LIN {X 0,Y 368.879,Z 269.346,A -85,B 0,C 180,E1 -12556.695,E2 -12556.695} C_VEL
LIN {X 0,Y 368.88,Z 269.35,A -85,B 0,C 180,E1 -12559.648,E2 -12559.648} C_VEL
LIN {X 0,Y 368.892,Z 269.345,A -85,B 0,C 180,E1 -12563.145,E2 -12563.145} C_VEL
LIN {X 0,Y 368.891,Z 269.344,A -85,B 0,C 180,E1 -12566.461,E2 -12566.461} C_VEL
LIN {X 0,Y 368.891,Z 269.346,A -85,B 0,C 180,E1 -12569.043,E2 -12569.043} C_VEL
LIN {X 0,Y 368.902,Z 269.348,A -85,B 0,C 180,E1 -12571.557,E2 -12571.557} C_VEL
LIN {X 0,Y 368.909,Z 269.347,A -85,B 0,C 180,E1 -12575.221,E2 -12575.221} C_VEL
LIN {X 0,Y 368.904,Z 269.344,A -85,B 0,C 180,E1 -12578.779,E2 -12578.779} C_VEL
LIN {X 0,Y 368.948,Z 269.337,A -85,B 0,C 180,E1 -12582.255,E2 -12582.255} C_VEL
LIN {X 0,Y 369.032,Z 269.327,A -85,B 0,C 180,E1 -12586.228,E2 -12586.228} C_VEL
LIN {X 0,Y 369.052,Z 269.324,A -85,B 0,C 180,E1 -12590.131,E2 -12590.131} C_VEL
LIN {X 0,Y 369.15,Z 269.313,A -85,B 0,C 180,E1 -12593.441,E2 -12593.441} C_VEL
LIN {X 0,Y 369.295,Z 269.294,A -85,B 0,C 180,E1 -12597.819,E2 -12597.819} C_VEL
LIN {X 0,Y 369.295,Z 269.297,A -85,B 0,C 180,E1 -12602.181,E2 -12602.181} C_VEL
LIN {X 0,Y 369.148,Z 269.316,A -85,B 0,C 180,E1 -12606.559,E2 -12606.559} C_VEL
LIN {X 0,Y 369.052,Z 269.326,A -85,B 0,C 180,E1 -12609.869,E2 -12609.869} C_VEL
LIN {X 0,Y 369.032,Z 269.329,A -85,B 0,C 180,E1 -12613.772,E2 -12613.772} C_VEL
LIN {X 0,Y 368.948,Z 269.34,A -85,B 0,C 180,E1 -12617.745,E2 -12617.745} C_VEL
LIN {X 0,Y 368.903,Z 269.343,A -85,B 0,C 180,E1 -12621.221,E2 -12621.221} C_VEL
LIN {X 0,Y 368.902,Z 269.348,A -85,B 0,C 180,E1 -12623.874,E2 -12623.874} C_VEL
LIN {X 0,Y 368.851,Z 269.35,A -85,B 0,C 180,E1 -12627.212,E2 -12627.212} C_VEL
LIN {X 0,Y 368.886,Z 269.35,A -85,B 0,C 180,E1 -12629.693,E2 -12629.693} C_VEL
LIN {X 0,Y 368.89,Z 269.345,A -85,B 0,C 180,E1 -12633.043,E2 -12633.043} C_VEL
LIN {X 0,Y 368.91,Z 269.342,A -85,B 0,C 180,E1 -12636.198,E2 -12636.198} C_VEL
LIN {X 0,Y 368.868,Z 269.349,A -85,B 0,C 180,E1 -12638.957,E2 -12638.957} C_VEL
LIN {X 0,Y 368.853,Z 269.349,A -85,B 0,C 180,E1 -12642.006,E2 -12642.006} C_VEL
LIN {X 0,Y 368.869,Z 269.353,A -85,B 0,C 180,E1 -12645.175,E2 -12645.175} C_VEL
LIN {X 0,Y 368.856,Z 269.348,A -85,B 0,C 180,E1 -12648.175,E2 -12648.175} C_VEL
LIN {X 0,Y 368.871,Z 269.349,A -85,B 0,C 180,E1 -12651.367,E2 -12651.367} C_VEL
LIN {X 0,Y 368.926,Z 269.343,A -85,B 0,C 180,E1 -12655.146,E2 -12655.146} C_VEL
LIN {X 0,Y 368.892,Z 269.347,A -85,B 0,C 180,E1 -12659.044,E2 -12659.044} C_VEL
LIN {X 0,Y 368.932,Z 269.441,A -85,B 0,C 180,E1 -12662.564,E2 -12662.564} C_VEL
LIN {X 0,Y 371.142,Z 280.964,A -85,B 0,C 180,E1 -12665.558,E2 -12665.558} C_VEL
LIN {X 0,Y 370.932,Z 287.523,A -85,B 0,C 180,E1 -12667.145,E2 -12667.145} C_VEL
LIN {X 0,Y 369.772,Z 303.185,A -85,B 0,C 180,E1 -12670.862,E2 -12670.862} C_VEL
LIN {X 0,Y 369.194,Z 312.035,A -85,B 0,C 180,E1 -12672.947,E2 -12672.947} C_VEL
LIN {X 0,Y 372.572,Z 338.491,A -85,B 0,C 180,E1 -12673.629,E2 -12673.629} C_VEL
LIN {X 0,Y 373.125,Z 345.859,A -85,B 0,C 180,E1 -12673.798,E2 -12673.798} C_VEL
LIN {X 0,Y 372.569,Z 389.778,A -85,B 0,C 180,E1 -12674.664,E2 -12674.664} C_VEL
LIN {X 0,Y 372.153,Z 399.376,A -85,B 0,C 180,E1 -12674.986,E2 -12674.986} C_VEL
LIN {X 0,Y 371.63,Z 409.413,A -85,B 0,C 180,E1 -12675.489,E2 -12675.489} C_VEL
LIN {X 0,Y 370.884,Z 420.823,A -85,B 0,C 180,E1 -12676.299,E2 -12676.299} C_VEL
LIN {X 0,Y 370.198,Z 429.423,A -85,B 0,C 180,E1 -12677.111,E2 -12677.111} C_VEL
LIN {X 0,Y 369.516,Z 437.52,A -85,B 0,C 180,E1 -12678.064,E2 -12678.064} C_VEL
LIN {X 0,Y 368.999,Z 444.218,A -85,B 0,C 180,E1 -12679.021,E2 -12679.021} C_VEL
LIN {X 0,Y 368.476,Z 450.579,A -85,B 0,C 180,E1 -12680.116,E2 -12680.116} C_VEL
LIN {X 0,Y 368.086,Z 455.87,A -85,B 0,C 180,E1 -12681.214,E2 -12681.214} C_VEL
LIN {X 0,Y 367.863,Z 460.289,A -85,B 0,C 180,E1 -12682.315,E2 -12682.315} C_VEL
LIN {X 0,Y 367.557,Z 465.239,A -85,B 0,C 180,E1 -12683.87,E2 -12683.87} C_VEL
LIN {X 0,Y 367.535,Z 468.17,A -85,B 0,C 180,E1 -12685.064,E2 -12685.064} C_VEL
LIN {X 0,Y 367.462,Z 471.098,A -85,B 0,C 180,E1 -12686.711,E2 -12686.711} C_VEL
LIN {X 0,Y 367.541,Z 472.367,A -85,B 0,C 180,E1 -12687.809,E2 -12687.809} C_VEL
LIN {X 0,Y 367.585,Z 473.154,A -85,B 0,C 180,E1 -12688.905,E2 -12688.905} C_VEL
LIN {X 0,Y 367.581,Z 473.451,A -85,B 0,C 180,E1 -12690.001,E2 -12690.001} C_VEL
LIN {X 0,Y 367.585,Z 473.151,A -85,B 0,C 180,E1 -12691.096,E2 -12691.096} C_VEL
LIN {X 0,Y 367.542,Z 472.355,A -85,B 0,C 180,E1 -12692.192,E2 -12692.192} C_VEL
LIN {X 0,Y 367.462,Z 471.079,A -85,B 0,C 180,E1 -12693.29,E2 -12693.29} C_VEL
LIN {X 0,Y 367.535,Z 468.144,A -85,B 0,C 180,E1 -12694.937,E2 -12694.937} C_VEL
LIN {X 0,Y 367.557,Z 465.207,A -85,B 0,C 180,E1 -12696.13,E2 -12696.13} C_VEL
LIN {X 0,Y 367.832,Z 460.241,A -85,B 0,C 180,E1 -12697.687,E2 -12697.687} C_VEL
LIN {X 0,Y 368.27,Z 453.362,A -85,B 0,C 180,E1 -12699.336,E2 -12699.336} C_VEL
LIN {X 0,Y 368.87,Z 445.856,A -85,B 0,C 180,E1 -12700.706,E2 -12700.706} C_VEL
LIN {X 0,Y 369.431,Z 438.457,A -85,B 0,C 180,E1 -12701.801,E2 -12701.801} C_VEL
LIN {X 0,Y 370.069,Z 430.542,A -85,B 0,C 180,E1 -12702.755,E2 -12702.755} C_VEL
LIN {X 0,Y 370.79,Z 422.188,A -85,B 0,C 180,E1 -12703.566,E2 -12703.566} C_VEL
LIN {X 0,Y 371.428,Z 411.508,A -85,B 0,C 180,E1 -12704.38,E2 -12704.38} C_VEL
LIN {X 0,Y 372.091,Z 399.889,A -85,B 0,C 180,E1 -12704.983,E2 -12704.983} C_VEL
LIN {X 0,Y 372.515,Z 390.149,A -85,B 0,C 180,E1 -12705.316,E2 -12705.316} C_VEL
LIN {X 0,Y 373.127,Z 345.225,A -85,B 0,C 180,E1 -12706.202,E2 -12706.202} C_VEL
LIN {X 0,Y 371.249,Z 327.242,A -85,B 0,C 180,E1 -12706.638,E2 -12706.638} C_VEL
LIN {X 0,Y 369.171,Z 312.021,A -85,B 0,C 180,E1 -12707.045,E2 -12707.045} C_VEL
LIN {X 0,Y 370.215,Z 297.109,A -85,B 0,C 180,E1 -12710.561,E2 -12710.561} C_VEL
LIN {X 0,Y 371.25,Z 282.618,A -85,B 0,C 180,E1 -12714.018,E2 -12714.018} C_VEL
LIN {X 0,Y 369.812,Z 273.814,A -85,B 0,C 180,E1 -12716.27,E2 -12716.27} C_VEL
LIN {X 0,Y 368.889,Z 269.349,A -85,B 0,C 180,E1 -12717.479,E2 -12717.479} C_VEL
LIN {X 0,Y 368.886,Z 269.348,A -85,B 0,C 180,E1 -12720.981,E2 -12720.981} C_VEL
LIN {X 0,Y 368.93,Z 269.342,A -85,B 0,C 180,E1 -12724.855,E2 -12724.855} C_VEL
LIN {X 0,Y 368.874,Z 269.348,A -85,B 0,C 180,E1 -12728.634,E2 -12728.634} C_VEL
LIN {X 0,Y 368.858,Z 269.348,A -85,B 0,C 180,E1 -12732.005,E2 -12732.005} C_VEL
LIN {X 0,Y 368.874,Z 269.348,A -85,B 0,C 180,E1 -12735.175,E2 -12735.175} C_VEL
LIN {X 0,Y 368.86,Z 269.349,A -85,B 0,C 180,E1 -12738.175,E2 -12738.175} C_VEL
LIN {X 0,Y 368.876,Z 269.346,A -85,B 0,C 180,E1 -12741.367,E2 -12741.367} C_VEL
LIN {X 0,Y 368.931,Z 269.34,A -85,B 0,C 180,E1 -12745.146,E2 -12745.146} C_VEL
LIN {X 0,Y 368.897,Z 269.344,A -85,B 0,C 180,E1 -12749.044,E2 -12749.044} C_VEL
LIN {X 0,Y 368.907,Z 269.342,A -85,B 0,C 180,E1 -12751.558,E2 -12751.558} C_VEL
LIN {X 0,Y 368.919,Z 269.344,A -85,B 0,C 180,E1 -12754.014,E2 -12754.014} C_VEL
LIN {X 0,Y 368.895,Z 269.345,A -85,B 0,C 180,E1 -12757.603,E2 -12757.603} C_VEL
LIN {X 0,Y 368.898,Z 269.343,A -85,B 0,C 180,E1 -12761.103,E2 -12761.103} C_VEL
LIN {X 0,Y 368.921,Z 269.341,A -85,B 0,C 180,E1 -12764.532,E2 -12764.532} C_VEL
LIN {X 0,Y 369.024,Z 269.327,A -85,B 0,C 180,E1 -12766.789,E2 -12766.789} C_VEL
LIN {X 0,Y 369.058,Z 269.326,A -85,B 0,C 180,E1 -12770.132,E2 -12770.132} C_VEL
LIN {X 0,Y 369.156,Z 269.315,A -85,B 0,C 180,E1 -12773.441,E2 -12773.441} C_VEL
LIN {X 0,Y 369.297,Z 269.297,A -85,B 0,C 180,E1 -12777.819,E2 -12777.819} C_VEL
LIN {X 0,Y 369.302,Z 269.293,A -85,B 0,C 180,E1 -12782.181,E2 -12782.181} C_VEL
LIN {X 0,Y 369.156,Z 269.312,A -85,B 0,C 180,E1 -12786.559,E2 -12786.559} C_VEL
LIN {X 0,Y 369.059,Z 269.324,A -85,B 0,C 180,E1 -12789.869,E2 -12789.869} C_VEL
LIN {X 0,Y 369.039,Z 269.326,A -85,B 0,C 180,E1 -12793.772,E2 -12793.772} C_VEL
LIN {X 0,Y 368.955,Z 269.336,A -85,B 0,C 180,E1 -12797.745,E2 -12797.745} C_VEL
LIN {X 0,Y 368.91,Z 269.344,A -85,B 0,C 180,E1 -12801.221,E2 -12801.221} C_VEL
LIN {X 0,Y 368.91,Z 269.342,A -85,B 0,C 180,E1 -12803.874,E2 -12803.874} C_VEL
LIN {X 0,Y 368.86,Z 269.349,A -85,B 0,C 180,E1 -12807.212,E2 -12807.212} C_VEL
LIN {X 0,Y 368.894,Z 269.344,A -85,B 0,C 180,E1 -12809.692,E2 -12809.692} C_VEL
LIN {X 0,Y 368.898,Z 269.344,A -85,B 0,C 180,E1 -12813.043,E2 -12813.043} C_VEL
LIN {X 0,Y 368.913,Z 269.346,A -85,B 0,C 180,E1 -12816.197,E2 -12816.197} C_VEL
LIN {X 0,Y 368.875,Z 269.347,A -85,B 0,C 180,E1 -12818.957,E2 -12818.957} C_VEL
LIN {X 0,Y 368.86,Z 269.352,A -85,B 0,C 180,E1 -12822.005,E2 -12822.005} C_VEL
LIN {X 0,Y 368.874,Z 269.346,A -85,B 0,C 180,E1 -12825.174,E2 -12825.174} C_VEL
LIN {X 0,Y 368.862,Z 269.352,A -85,B 0,C 180,E1 -12828.174,E2 -12828.174} C_VEL
LIN {X 0,Y 368.879,Z 269.347,A -85,B 0,C 180,E1 -12831.366,E2 -12831.366} C_VEL
LIN {X 0,Y 368.933,Z 269.34,A -85,B 0,C 180,E1 -12835.146,E2 -12835.146} C_VEL
LIN {X 0,Y 368.897,Z 269.344,A -85,B 0,C 180,E1 -12839.043,E2 -12839.043} C_VEL
LIN {X 0,Y 368.908,Z 269.347,A -85,B 0,C 180,E1 -12841.557,E2 -12841.557} C_VEL
LIN {X 0,Y 368.916,Z 269.345,A -85,B 0,C 180,E1 -12845.221,E2 -12845.221} C_VEL
LIN {X 0,Y 368.912,Z 269.343,A -85,B 0,C 180,E1 -12848.779,E2 -12848.779} C_VEL
LIN {X 0,Y 368.942,Z 269.431,A -85,B 0,C 180,E1 -12851.867,E2 -12851.867} C_VEL
LIN {X 0,Y 369.672,Z 273.533,A -85,B 0,C 180,E1 -12853.03,E2 -12853.03} C_VEL
LIN {X 0,Y 371.877,Z 282.5,A -85,B 0,C 180,E1 -12853.328,E2 -12853.328} C_VEL
LIN {X 0,Y 373.696,Z 292.657,A -85,B 0,C 180,E1 -12853.614,E2 -12853.614} C_VEL
LIN {X 0,Y 372.903,Z 350.075,A -85,B 0,C 180,E1 -12854.736,E2 -12854.736} C_VEL
LIN {X 0,Y 372.721,Z 359.09,A -85,B 0,C 180,E1 -12855.043,E2 -12855.043} C_VEL
LIN {X 0,Y 372.44,Z 368.63,A -85,B 0,C 180,E1 -12855.52,E2 -12855.52} C_VEL
LIN {X 0,Y 371.918,Z 378.632,A -85,B 0,C 180,E1 -12856.197,E2 -12856.197} C_VEL
LIN {X 0,Y 371.346,Z 388.997,A -85,B 0,C 180,E1 -12857.151,E2 -12857.151} C_VEL
LIN {X 0,Y 370.731,Z 397.111,A -85,B 0,C 180,E1 -12858.102,E2 -12858.102} C_VEL
LIN {X 0,Y 370.172,Z 403.801,A -85,B 0,C 180,E1 -12859.055,E2 -12859.055} C_VEL
LIN {X 0,Y 369.607,Z 410.133,A -85,B 0,C 180,E1 -12860.146,E2 -12860.146} C_VEL
LIN {X 0,Y 369.036,Z 416.557,A -85,B 0,C 180,E1 -12861.512,E2 -12861.512} C_VEL
LIN {X 0,Y 368.588,Z 422.411,A -85,B 0,C 180,E1 -12863.094,E2 -12863.094} C_VEL
LIN {X 0,Y 368.154,Z 426.418,A -85,B 0,C 180,E1 -12864.522,E2 -12864.522} C_VEL
LIN {X 0,Y 368.033,Z 428.723,A -85,B 0,C 180,E1 -12865.619,E2 -12865.619} C_VEL
LIN {X 0,Y 367.918,Z 430.478,A -85,B 0,C 180,E1 -12866.714,E2 -12866.714} C_VEL
LIN {X 0,Y 367.735,Z 431.749,A -85,B 0,C 180,E1 -12867.809,E2 -12867.809} C_VEL
LIN {X 0,Y 367.62,Z 432.553,A -85,B 0,C 180,E1 -12868.904,E2 -12868.904} C_VEL
LIN {X 0,Y 367.588,Z 432.858,A -85,B 0,C 180,E1 -12869.999,E2 -12869.999} C_VEL
LIN {X 0,Y 367.62,Z 432.583,A -85,B 0,C 180,E1 -12871.095,E2 -12871.095} C_VEL
LIN {X 0,Y 367.733,Z 431.84,A -85,B 0,C 180,E1 -12872.19,E2 -12872.19} C_VEL
LIN {X 0,Y 367.913,Z 430.63,A -85,B 0,C 180,E1 -12873.285,E2 -12873.285} C_VEL
LIN {X 0,Y 368.112,Z 427.798,A -85,B 0,C 180,E1 -12874.928,E2 -12874.928} C_VEL
LIN {X 0,Y 368.265,Z 425.223,A -85,B 0,C 180,E1 -12876.024,E2 -12876.024} C_VEL
LIN {X 0,Y 368.848,Z 419.753,A -85,B 0,C 180,E1 -12877.776,E2 -12877.776} C_VEL
LIN {X 0,Y 369.31,Z 413.463,A -85,B 0,C 180,E1 -12879.308,E2 -12879.308} C_VEL
LIN {X 0,Y 369.986,Z 406.124,A -85,B 0,C 180,E1 -12880.672,E2 -12880.672} C_VEL
LIN {X 0,Y 370.696,Z 398.874,A -85,B 0,C 180,E1 -12881.759,E2 -12881.759} C_VEL
LIN {X 0,Y 371.137,Z 392.354,A -85,B 0,C 180,E1 -12882.577,E2 -12882.577} C_VEL
LIN {X 0,Y 371.625,Z 384.454,A -85,B 0,C 180,E1 -12883.395,E2 -12883.395} C_VEL
LIN {X 0,Y 372.128,Z 376.286,A -85,B 0,C 180,E1 -12884.072,E2 -12884.072} C_VEL
LIN {X 0,Y 372.549,Z 368.006,A -85,B 0,C 180,E1 -12884.614,E2 -12884.614} C_VEL
LIN {X 0,Y 372.752,Z 359.066,A -85,B 0,C 180,E1 -12885.06,E2 -12885.06} C_VEL
LIN {X 0,Y 372.943,Z 350.249,A -85,B 0,C 180,E1 -12885.361,E2 -12885.361} C_VEL
LIN {X 0,Y 373.415,Z 319.78,A -85,B 0,C 180,E1 -12885.969,E2 -12885.969} C_VEL
LIN {X 0,Y 372.594,Z 312.039,A -85,B 0,C 180,E1 -12886.158,E2 -12886.158} C_VEL
LIN {X 0,Y 370.77,Z 304.493,A -85,B 0,C 180,E1 -12886.391,E2 -12886.391} C_VEL
LIN {X 0,Y 366.304,Z 289.542,A -85,B 0,C 180,E1 -12886.902,E2 -12886.902} C_VEL
LIN {X 0,Y 363.598,Z 277.387,A -85,B 0,C 180,E1 -12887.282,E2 -12887.282} C_VEL
LIN {X 0,Y 362.549,Z 273.87,A -85,B 0,C 180,E1 -12887.437,E2 -12887.437} C_VEL
LIN {X 0,Y 361.902,Z 270.219,A -85,B 0,C 180,E1 -12888.541,E2 -12888.541} C_VEL
LIN {X 0,Y 361.858,Z 270.22,A -85,B 0,C 180,E1 -12891.654,E2 -12891.654} C_VEL
LIN {X 0,Y 361.858,Z 270.22,A -85,B 0,C 180,E1 -12895.294,E2 -12895.294} C_VEL
LIN {X 0,Y 361.854,Z 270.221,A -85,B 0,C 180,E1 -12899.073,E2 -12899.073} C_VEL
LIN {X 0,Y 361.844,Z 270.223,A -85,B 0,C 180,E1 -12902.944,E2 -12902.944} C_VEL
LIN {X 0,Y 361.861,Z 270.22,A -85,B 0,C 180,E1 -12905.637,E2 -12905.637} C_VEL
LIN {X 0,Y 361.823,Z 270.224,A -85,B 0,C 180,E1 -12909.017,E2 -12909.017} C_VEL
LIN {X 0,Y 361.825,Z 270.224,A -85,B 0,C 180,E1 -12912.829,E2 -12912.829} C_VEL
LIN {X 0,Y 361.809,Z 270.231,A -85,B 0,C 180,E1 -12915.947,E2 -12915.947} C_VEL
LIN {X 0,Y 361.806,Z 270.228,A -85,B 0,C 180,E1 -12919.249,E2 -12919.249} C_VEL
LIN {X 0,Y 361.858,Z 270.22,A -85,B 0,C 180,E1 -12922.981,E2 -12922.981} C_VEL
LIN {X 0,Y 361.853,Z 270.221,A -85,B 0,C 180,E1 -12926.631,E2 -12926.631} C_VEL
LIN {X 0,Y 361.842,Z 270.227,A -85,B 0,C 180,E1 -12929.669,E2 -12929.669} C_VEL
LIN {X 0,Y 361.851,Z 270.226,A -85,B 0,C 180,E1 -12933.467,E2 -12933.467} C_VEL
LIN {X 0,Y 361.871,Z 270.223,A -85,B 0,C 180,E1 -12937.143,E2 -12937.143} C_VEL
LIN {X 0,Y 361.85,Z 270.223,A -85,B 0,C 180,E1 -12940.72,E2 -12940.72} C_VEL
LIN {X 0,Y 361.89,Z 270.216,A -85,B 0,C 180,E1 -12944.223,E2 -12944.223} C_VEL
LIN {X 0,Y 361.994,Z 270.205,A -85,B 0,C 180,E1 -12946.527,E2 -12946.527} C_VEL
LIN {X 0,Y 361.989,Z 270.204,A -85,B 0,C 180,E1 -12949.937,E2 -12949.937} C_VEL
LIN {X 0,Y 362.114,Z 270.19,A -85,B 0,C 180,E1 -12953.313,E2 -12953.313} C_VEL
LIN {X 0,Y 362.258,Z 270.17,A -85,B 0,C 180,E1 -12957.776,E2 -12957.776} C_VEL
LIN {X 0,Y 362.168,Z 270.183,A -85,B 0,C 180,E1 -12961.112,E2 -12961.112} C_VEL
LIN {X 0,Y 362.258,Z 270.173,A -85,B 0,C 180,E1 -12962.224,E2 -12962.224} C_VEL
LIN {X 0,Y 362.112,Z 270.191,A -85,B 0,C 180,E1 -12966.687,E2 -12966.687} C_VEL
LIN {X 0,Y 361.989,Z 270.208,A -85,B 0,C 180,E1 -12970.063,E2 -12970.063} C_VEL
LIN {X 0,Y 361.974,Z 270.209,A -85,B 0,C 180,E1 -12973.887,E2 -12973.887} C_VEL
LIN {X 0,Y 361.879,Z 270.223,A -85,B 0,C 180,E1 -12978.103,E2 -12978.103} C_VEL
LIN {X 0,Y 361.847,Z 270.225,A -85,B 0,C 180,E1 -12981.656,E2 -12981.656} C_VEL
LIN {X 0,Y 361.846,Z 270.223,A -85,B 0,C 180,E1 -12985.296,E2 -12985.296} C_VEL
LIN {X 0,Y 361.85,Z 270.222,A -85,B 0,C 180,E1 -12989.074,E2 -12989.074} C_VEL
LIN {X 0,Y 361.842,Z 270.223,A -85,B 0,C 180,E1 -12992.945,E2 -12992.945} C_VEL
LIN {X 0,Y 361.861,Z 270.224,A -85,B 0,C 180,E1 -12995.637,E2 -12995.637} C_VEL
LIN {X 0,Y 361.82,Z 270.227,A -85,B 0,C 180,E1 -12999.018,E2 -12999.018} C_VEL
LIN {X 0,Y 361.824,Z 270.226,A -85,B 0,C 180,E1 -13002.83,E2 -13002.83} C_VEL
LIN {X 0,Y 361.808,Z 270.226,A -85,B 0,C 180,E1 -13005.948,E2 -13005.948} C_VEL
LIN {X 0,Y 361.806,Z 270.231,A -85,B 0,C 180,E1 -13009.25,E2 -13009.25} C_VEL
LIN {X 0,Y 361.857,Z 270.226,A -85,B 0,C 180,E1 -13012.982,E2 -13012.982} C_VEL
LIN {X 0,Y 361.853,Z 270.224,A -85,B 0,C 180,E1 -13016.632,E2 -13016.632} C_VEL
LIN {X 0,Y 361.843,Z 270.221,A -85,B 0,C 180,E1 -13019.67,E2 -13019.67} C_VEL
LIN {X 0,Y 361.88,Z 270.344,A -85,B 0,C 180,E1 -13022.323,E2 -13022.323} C_VEL
LIN {X 0,Y 363.955,Z 281.06,A -85,B 0,C 180,E1 -13025.172,E2 -13025.172} C_VEL
LIN {X 0,Y 364.21,Z 284.703,A -85,B 0,C 180,E1 -13026.095,E2 -13026.095} C_VEL
LIN {X 0,Y 363.046,Z 300.385,A -85,B 0,C 180,E1 -13029.904,E2 -13029.904} C_VEL
LIN {X 0,Y 362.237,Z 311.635,A -85,B 0,C 180,E1 -13032.609,E2 -13032.609} C_VEL
LIN {X 0,Y 365.874,Z 340.177,A -85,B 0,C 180,E1 -13033.362,E2 -13033.362} C_VEL
LIN {X 0,Y 366.3,Z 346.247,A -85,B 0,C 180,E1 -13033.503,E2 -13033.503} C_VEL
LIN {X 0,Y 365.733,Z 389.456,A -85,B 0,C 180,E1 -13034.372,E2 -13034.372} C_VEL
LIN {X 0,Y 365.302,Z 398.993,A -85,B 0,C 180,E1 -13034.697,E2 -13034.697} C_VEL
LIN {X 0,Y 364.761,Z 409.028,A -85,B 0,C 180,E1 -13035.21,E2 -13035.21} C_VEL
LIN {X 0,Y 363.98,Z 420.435,A -85,B 0,C 180,E1 -13036.034,E2 -13036.034} C_VEL
LIN {X 0,Y 363.251,Z 429.033,A -85,B 0,C 180,E1 -13036.861,E2 -13036.861} C_VEL
LIN {X 0,Y 362.554,Z 437.13,A -85,B 0,C 180,E1 -13037.831,E2 -13037.831} C_VEL
LIN {X 0,Y 361.995,Z 443.826,A -85,B 0,C 180,E1 -13038.806,E2 -13038.806} C_VEL
LIN {X 0,Y 361.447,Z 450.187,A -85,B 0,C 180,E1 -13039.922,E2 -13039.922} C_VEL
LIN {X 0,Y 361.056,Z 455.478,A -85,B 0,C 180,E1 -13041.042,E2 -13041.042} C_VEL
LIN {X 0,Y 360.788,Z 459.897,A -85,B 0,C 180,E1 -13042.164,E2 -13042.164} C_VEL
LIN {X 0,Y 360.481,Z 465.205,A -85,B 0,C 180,E1 -13043.88,E2 -13043.88} C_VEL
LIN {X 0,Y 360.45,Z 468.946,A -85,B 0,C 180,E1 -13045.527,E2 -13045.527} C_VEL
LIN {X 0,Y 360.379,Z 470.707,A -85,B 0,C 180,E1 -13046.647,E2 -13046.647} C_VEL
LIN {X 0,Y 360.442,Z 471.975,A -85,B 0,C 180,E1 -13047.766,E2 -13047.766} C_VEL
LIN {X 0,Y 360.519,Z 472.764,A -85,B 0,C 180,E1 -13048.884,E2 -13048.884} C_VEL
LIN {X 0,Y 360.515,Z 473.06,A -85,B 0,C 180,E1 -13050.001,E2 -13050.001} C_VEL
LIN {X 0,Y 360.519,Z 472.76,A -85,B 0,C 180,E1 -13051.118,E2 -13051.118} C_VEL
LIN {X 0,Y 360.442,Z 471.963,A -85,B 0,C 180,E1 -13052.235,E2 -13052.235} C_VEL
LIN {X 0,Y 360.379,Z 470.687,A -85,B 0,C 180,E1 -13053.355,E2 -13053.355} C_VEL
LIN {X 0,Y 360.447,Z 467.75,A -85,B 0,C 180,E1 -13055.034,E2 -13055.034} C_VEL
LIN {X 0,Y 360.482,Z 465.171,A -85,B 0,C 180,E1 -13056.12,E2 -13056.12} C_VEL
LIN {X 0,Y 360.763,Z 459.846,A -85,B 0,C 180,E1 -13057.838,E2 -13057.838} C_VEL
LIN {X 0,Y 361.215,Z 452.965,A -85,B 0,C 180,E1 -13059.52,E2 -13059.52} C_VEL
LIN {X 0,Y 361.878,Z 445.461,A -85,B 0,C 180,E1 -13060.916,E2 -13060.916} C_VEL
LIN {X 0,Y 362.472,Z 438.062,A -85,B 0,C 180,E1 -13062.031,E2 -13062.031} C_VEL
LIN {X 0,Y 363.148,Z 430.147,A -85,B 0,C 180,E1 -13063.002,E2 -13063.002} C_VEL
LIN {X 0,Y 363.892,Z 421.792,A -85,B 0,C 180,E1 -13063.828,E2 -13063.828} C_VEL
LIN {X 0,Y 364.56,Z 411.111,A -85,B 0,C 180,E1 -13064.657,E2 -13064.657} C_VEL
LIN {X 0,Y 365.229,Z 399.487,A -85,B 0,C 180,E1 -13065.272,E2 -13065.272} C_VEL
LIN {X 0,Y 365.681,Z 389.743,A -85,B 0,C 180,E1 -13065.609,E2 -13065.609} C_VEL
LIN {X 0,Y 366.191,Z 352.168,A -85,B 0,C 180,E1 -13066.37,E2 -13066.37} C_VEL
LIN {X 0,Y 366.184,Z 343.057,A -85,B 0,C 180,E1 -13066.553,E2 -13066.553} C_VEL
LIN {X 0,Y 362.894,Z 316.548,A -85,B 0,C 180,E1 -13067.239,E2 -13067.239} C_VEL
LIN {X 0,Y 362.207,Z 311.616,A -85,B 0,C 180,E1 -13067.383,E2 -13067.383} C_VEL
LIN {X 0,Y 363.286,Z 296.707,A -85,B 0,C 180,E1 -13070.971,E2 -13070.971} C_VEL
LIN {X 0,Y 364.256,Z 284.637,A -85,B 0,C 180,E1 -13073.903,E2 -13073.903} C_VEL
LIN {X 0,Y 363.496,Z 278.509,A -85,B 0,C 180,E1 -13075.48,E2 -13075.48} C_VEL
LIN {X 0,Y 361.849,Z 270.225,A -85,B 0,C 180,E1 -13077.721,E2 -13077.721} C_VEL
LIN {X 0,Y 361.827,Z 270.229,A -85,B 0,C 180,E1 -13081.28,E2 -13081.28} C_VEL
LIN {X 0,Y 361.85,Z 270.221,A -85,B 0,C 180,E1 -13084.281,E2 -13084.281} C_VEL
LIN {X 0,Y 361.856,Z 270.224,A -85,B 0,C 180,E1 -13087.221,E2 -13087.221} C_VEL
LIN {X 0,Y 361.811,Z 270.23,A -85,B 0,C 180,E1 -13090.751,E2 -13090.751} C_VEL
LIN {X 0,Y 361.812,Z 270.227,A -85,B 0,C 180,E1 -13094.37,E2 -13094.37} C_VEL
LIN {X 0,Y 361.823,Z 270.224,A -85,B 0,C 180,E1 -13097.571,E2 -13097.571} C_VEL
LIN {X 0,Y 361.842,Z 270.222,A -85,B 0,C 180,E1 -13101.572,E2 -13101.572} C_VEL
LIN {X 0,Y 361.87,Z 270.223,A -85,B 0,C 180,E1 -13104.657,E2 -13104.657} C_VEL
LIN {X 0,Y 361.838,Z 270.228,A -85,B 0,C 180,E1 -13108.371,E2 -13108.371} C_VEL
LIN {X 0,Y 361.85,Z 270.222,A -85,B 0,C 180,E1 -13110.951,E2 -13110.951} C_VEL
LIN {X 0,Y 361.852,Z 270.222,A -85,B 0,C 180,E1 -13114.704,E2 -13114.704} C_VEL
LIN {X 0,Y 361.853,Z 270.224,A -85,B 0,C 180,E1 -13118.345,E2 -13118.345} C_VEL
LIN {X 0,Y 361.896,Z 270.22,A -85,B 0,C 180,E1 -13122.098,E2 -13122.098} C_VEL
LIN {X 0,Y 361.952,Z 270.212,A -85,B 0,C 180,E1 -13126.132,E2 -13126.132} C_VEL
LIN {X 0,Y 361.994,Z 270.207,A -85,B 0,C 180,E1 -13129.937,E2 -13129.937} C_VEL
LIN {X 0,Y 362.121,Z 270.19,A -85,B 0,C 180,E1 -13133.313,E2 -13133.313} C_VEL
LIN {X 0,Y 362.259,Z 270.174,A -85,B 0,C 180,E1 -13137.776,E2 -13137.776} C_VEL
LIN {X 0,Y 362.175,Z 270.184,A -85,B 0,C 180,E1 -13141.112,E2 -13141.112} C_VEL
LIN {X 0,Y 362.264,Z 270.169,A -85,B 0,C 180,E1 -13142.224,E2 -13142.224} C_VEL
LIN {X 0,Y 362.12,Z 270.189,A -85,B 0,C 180,E1 -13146.687,E2 -13146.687} C_VEL
LIN {X 0,Y 361.996,Z 270.203,A -85,B 0,C 180,E1 -13150.063,E2 -13150.063} C_VEL
LIN {X 0,Y 361.982,Z 270.205,A -85,B 0,C 180,E1 -13153.887,E2 -13153.887} C_VEL
LIN {X 0,Y 361.886,Z 270.217,A -85,B 0,C 180,E1 -13158.103,E2 -13158.103} C_VEL
LIN {X 0,Y 361.854,Z 270.221,A -85,B 0,C 180,E1 -13161.655,E2 -13161.655} C_VEL
LIN {X 0,Y 361.862,Z 270.22,A -85,B 0,C 180,E1 -13165.295,E2 -13165.295} C_VEL
LIN {X 0,Y 361.857,Z 270.222,A -85,B 0,C 180,E1 -13169.074,E2 -13169.074} C_VEL
LIN {X 0,Y 361.848,Z 270.223,A -85,B 0,C 180,E1 -13172.945,E2 -13172.945} C_VEL
LIN {X 0,Y 361.866,Z 270.219,A -85,B 0,C 180,E1 -13175.637,E2 -13175.637} C_VEL
LIN {X 0,Y 361.827,Z 270.224,A -85,B 0,C 180,E1 -13179.018,E2 -13179.018} C_VEL
LIN {X 0,Y 361.83,Z 270.224,A -85,B 0,C 180,E1 -13182.83,E2 -13182.83} C_VEL
LIN {X 0,Y 361.815,Z 270.23,A -85,B 0,C 180,E1 -13185.947,E2 -13185.947} C_VEL
LIN {X 0,Y 361.811,Z 270.226,A -85,B 0,C 180,E1 -13189.249,E2 -13189.249} C_VEL
LIN {X 0,Y 361.864,Z 270.219,A -85,B 0,C 180,E1 -13192.981,E2 -13192.981} C_VEL
LIN {X 0,Y 361.859,Z 270.22,A -85,B 0,C 180,E1 -13196.631,E2 -13196.631} C_VEL
LIN {X 0,Y 361.849,Z 270.227,A -85,B 0,C 180,E1 -13199.669,E2 -13199.669} C_VEL
LIN {X 0,Y 361.858,Z 270.226,A -85,B 0,C 180,E1 -13203.467,E2 -13203.467} C_VEL
LIN {X 0,Y 361.878,Z 270.221,A -85,B 0,C 180,E1 -13207.143,E2 -13207.143} C_VEL
LIN {X 0,Y 361.861,Z 270.229,A -85,B 0,C 180,E1 -13210.72,E2 -13210.72} C_VEL
LIN {X 0,Y 361.917,Z 270.316,A -85,B 0,C 180,E1 -13211.642,E2 -13211.642} C_VEL
LIN {X 0,Y 362.569,Z 274.019,A -85,B 0,C 180,E1 -13212.703,E2 -13212.703} C_VEL
LIN {X 0,Y 364.981,Z 282.896,A -85,B 0,C 180,E1 -13213.003,E2 -13213.003} C_VEL
LIN {X 0,Y 366.912,Z 293.073,A -85,B 0,C 180,E1 -13213.302,E2 -13213.302} C_VEL
LIN {X 0,Y 366.087,Z 350.483,A -85,B 0,C 180,E1 -13214.444,E2 -13214.444} C_VEL
LIN {X 0,Y 365.89,Z 359.492,A -85,B 0,C 180,E1 -13214.757,E2 -13214.757} C_VEL
LIN {X 0,Y 365.603,Z 369.028,A -85,B 0,C 180,E1 -13215.243,E2 -13215.243} C_VEL
LIN {X 0,Y 365.064,Z 379.029,A -85,B 0,C 180,E1 -13215.933,E2 -13215.933} C_VEL
LIN {X 0,Y 364.448,Z 389.392,A -85,B 0,C 180,E1 -13216.903,E2 -13216.903} C_VEL
LIN {X 0,Y 363.817,Z 397.505,A -85,B 0,C 180,E1 -13217.873,E2 -13217.873} C_VEL
LIN {X 0,Y 363.232,Z 404.195,A -85,B 0,C 180,E1 -13218.843,E2 -13218.843} C_VEL
LIN {X 0,Y 362.644,Z 410.526,A -85,B 0,C 180,E1 -13219.955,E2 -13219.955} C_VEL
LIN {X 0,Y 362.027,Z 416.95,A -85,B 0,C 180,E1 -13221.346,E2 -13221.346} C_VEL
LIN {X 0,Y 361.62,Z 422.028,A -85,B 0,C 180,E1 -13222.73,E2 -13222.73} C_VEL
LIN {X 0,Y 361.106,Z 426.811,A -85,B 0,C 180,E1 -13224.415,E2 -13224.415} C_VEL
LIN {X 0,Y 360.961,Z 429.115,A -85,B 0,C 180,E1 -13225.533,E2 -13225.533} C_VEL
LIN {X 0,Y 360.849,Z 430.87,A -85,B 0,C 180,E1 -13226.65,E2 -13226.65} C_VEL
LIN {X 0,Y 360.678,Z 432.14,A -85,B 0,C 180,E1 -13227.766,E2 -13227.766} C_VEL
LIN {X 0,Y 360.556,Z 432.943,A -85,B 0,C 180,E1 -13228.883,E2 -13228.883} C_VEL
LIN {X 0,Y 360.521,Z 433.248,A -85,B 0,C 180,E1 -13229.999,E2 -13229.999} C_VEL
LIN {X 0,Y 360.556,Z 432.973,A -85,B 0,C 180,E1 -13231.116,E2 -13231.116} C_VEL
LIN {X 0,Y 360.676,Z 432.229,A -85,B 0,C 180,E1 -13232.233,E2 -13232.233} C_VEL
LIN {X 0,Y 360.844,Z 431.02,A -85,B 0,C 180,E1 -13233.349,E2 -13233.349} C_VEL
LIN {X 0,Y 361.035,Z 428.19,A -85,B 0,C 180,E1 -13235.025,E2 -13235.025} C_VEL
LIN {X 0,Y 361.233,Z 425.612,A -85,B 0,C 180,E1 -13236.142,E2 -13236.142} C_VEL
LIN {X 0,Y 361.789,Z 420.526,A -85,B 0,C 180,E1 -13237.815,E2 -13237.815} C_VEL
LIN {X 0,Y 362.203,Z 415.061,A -85,B 0,C 180,E1 -13239.211,E2 -13239.211} C_VEL
LIN {X 0,Y 362.876,Z 408.184,A -85,B 0,C 180,E1 -13240.602,E2 -13240.602} C_VEL
LIN {X 0,Y 363.652,Z 400.278,A -85,B 0,C 180,E1 -13241.849,E2 -13241.849} C_VEL
LIN {X 0,Y 364.226,Z 392.741,A -85,B 0,C 180,E1 -13242.82,E2 -13242.82} C_VEL
LIN {X 0,Y 364.754,Z 384.839,A -85,B 0,C 180,E1 -13243.652,E2 -13243.652} C_VEL
LIN {X 0,Y 365.266,Z 376.67,A -85,B 0,C 180,E1 -13244.342,E2 -13244.342} C_VEL
LIN {X 0,Y 365.717,Z 368.388,A -85,B 0,C 180,E1 -13244.893,E2 -13244.893} C_VEL
LIN {X 0,Y 365.932,Z 359.444,A -85,B 0,C 180,E1 -13245.347,E2 -13245.347} C_VEL
LIN {X 0,Y 366.135,Z 349.57,A -85,B 0,C 180,E1 -13245.683,E2 -13245.683} C_VEL
LIN {X 0,Y 366.81,Z 292.25,A -85,B 0,C 180,E1 -13246.823,E2 -13246.823} C_VEL
LIN {X 0,Y 366.304,Z 289.542,A -85,B 0,C 180,E1 -13246.902,E2 -13246.902} C_VEL
LIN {X 0,Y 364.182,Z 284.497,A -85,B 0,C 180,E1 -13247.118,E2 -13247.118} C_VEL
LIN {X 0,Y 360.972,Z 280.063,A -85,B 0,C 180,E1 -13247.359,E2 -13247.359} C_VEL
LIN {X 0,Y 356.657,Z 275.394,A -85,B 0,C 180,E1 -13247.714,E2 -13247.714} C_VEL
LIN {X 0,Y 355.32,Z 273.431,A -85,B 0,C 180,E1 -13248.052,E2 -13248.052} C_VEL
LIN {X 0,Y 355.217,Z 273.11,A -85,B 0,C 180,E1 -13248.138,E2 -13248.138} C_VEL
LIN {X 0,Y 354.842,Z 271.1,A -85,B 0,C 180,E1 -13248.774,E2 -13248.774} C_VEL
LIN {X 0,Y 354.812,Z 271.099,A -85,B 0,C 180,E1 -13252.107,E2 -13252.107} C_VEL
LIN {X 0,Y 354.798,Z 271.1,A -85,B 0,C 180,E1 -13255.835,E2 -13255.835} C_VEL
LIN {X 0,Y 354.791,Z 271.1,A -85,B 0,C 180,E1 -13259.683,E2 -13259.683} C_VEL
LIN {X 0,Y 354.805,Z 271.099,A -85,B 0,C 180,E1 -13263.701,E2 -13263.701} C_VEL
LIN {X 0,Y 354.791,Z 271.104,A -85,B 0,C 180,E1 -13266.459,E2 -13266.459} C_VEL
LIN {X 0,Y 354.765,Z 271.104,A -85,B 0,C 180,E1 -13269.412,E2 -13269.412} C_VEL
LIN {X 0,Y 354.777,Z 271.102,A -85,B 0,C 180,E1 -13272.865,E2 -13272.865} C_VEL
LIN {X 0,Y 354.759,Z 271.109,A -85,B 0,C 180,E1 -13276.102,E2 -13276.102} C_VEL
LIN {X 0,Y 354.758,Z 271.105,A -85,B 0,C 180,E1 -13279.175,E2 -13279.175} C_VEL
LIN {X 0,Y 354.795,Z 271.1,A -85,B 0,C 180,E1 -13282.404,E2 -13282.404} C_VEL
LIN {X 0,Y 354.804,Z 271.099,A -85,B 0,C 180,E1 -13284.94,E2 -13284.94} C_VEL
LIN {X 0,Y 354.785,Z 271.101,A -85,B 0,C 180,E1 -13288.406,E2 -13288.406} C_VEL
LIN {X 0,Y 354.792,Z 271.105,A -85,B 0,C 180,E1 -13291.614,E2 -13291.614} C_VEL
LIN {X 0,Y 354.836,Z 271.1,A -85,B 0,C 180,E1 -13295.422,E2 -13295.422} C_VEL
LIN {X 0,Y 354.816,Z 271.102,A -85,B 0,C 180,E1 -13299.112,E2 -13299.112} C_VEL
LIN {X 0,Y 354.847,Z 271.095,A -85,B 0,C 180,E1 -13302.717,E2 -13302.717} C_VEL
LIN {X 0,Y 354.934,Z 271.083,A -85,B 0,C 180,E1 -13306.254,E2 -13306.254} C_VEL
LIN {X 0,Y 354.946,Z 271.081,A -85,B 0,C 180,E1 -13309.735,E2 -13309.735} C_VEL
LIN {X 0,Y 355.08,Z 271.067,A -85,B 0,C 180,E1 -13313.18,E2 -13313.18} C_VEL
LIN {X 0,Y 355.22,Z 271.047,A -85,B 0,C 180,E1 -13317.732,E2 -13317.732} C_VEL
LIN {X 0,Y 355.139,Z 271.058,A -85,B 0,C 180,E1 -13321.134,E2 -13321.134} C_VEL
LIN {X 0,Y 355.22,Z 271.05,A -85,B 0,C 180,E1 -13322.268,E2 -13322.268} C_VEL
LIN {X 0,Y 355.079,Z 271.066,A -85,B 0,C 180,E1 -13326.82,E2 -13326.82} C_VEL
LIN {X 0,Y 354.945,Z 271.087,A -85,B 0,C 180,E1 -13330.265,E2 -13330.265} C_VEL
LIN {X 0,Y 354.918,Z 271.089,A -85,B 0,C 180,E1 -13334.006,E2 -13334.006} C_VEL
LIN {X 0,Y 354.836,Z 271.1,A -85,B 0,C 180,E1 -13338.068,E2 -13338.068} C_VEL
LIN {X 0,Y 354.8,Z 271.103,A -85,B 0,C 180,E1 -13342.108,E2 -13342.108} C_VEL
LIN {X 0,Y 354.789,Z 271.106,A -85,B 0,C 180,E1 -13345.836,E2 -13345.836} C_VEL
LIN {X 0,Y 354.787,Z 271.106,A -85,B 0,C 180,E1 -13349.685,E2 -13349.685} C_VEL
LIN {X 0,Y 354.781,Z 271.102,A -85,B 0,C 180,E1 -13352.334,E2 -13352.334} C_VEL
LIN {X 0,Y 354.816,Z 271.101,A -85,B 0,C 180,E1 -13355.699,E2 -13355.699} C_VEL
LIN {X 0,Y 354.763,Z 271.109,A -85,B 0,C 180,E1 -13359.413,E2 -13359.413} C_VEL
LIN {X 0,Y 354.776,Z 271.104,A -85,B 0,C 180,E1 -13362.866,E2 -13362.866} C_VEL
LIN {X 0,Y 354.758,Z 271.104,A -85,B 0,C 180,E1 -13366.103,E2 -13366.103} C_VEL
LIN {X 0,Y 354.759,Z 271.109,A -85,B 0,C 180,E1 -13369.176,E2 -13369.176} C_VEL
LIN {X 0,Y 354.794,Z 271.101,A -85,B 0,C 180,E1 -13372.405,E2 -13372.405} C_VEL
LIN {X 0,Y 354.804,Z 271.104,A -85,B 0,C 180,E1 -13374.941,E2 -13374.941} C_VEL
LIN {X 0,Y 354.772,Z 271.105,A -85,B 0,C 180,E1 -13378.41,E2 -13378.41} C_VEL
LIN {X 0,Y 354.835,Z 271.199,A -85,B 0,C 180,E1 -13382.061,E2 -13382.061} C_VEL
LIN {X 0,Y 357.006,Z 282.399,A -85,B 0,C 180,E1 -13385.102,E2 -13385.102} C_VEL
LIN {X 0,Y 357.235,Z 285.51,A -85,B 0,C 180,E1 -13385.908,E2 -13385.908} C_VEL
LIN {X 0,Y 356.114,Z 299.985,A -85,B 0,C 180,E1 -13389.495,E2 -13389.495} C_VEL
LIN {X 0,Y 355.273,Z 311.205,A -85,B 0,C 180,E1 -13392.249,E2 -13392.249} C_VEL
LIN {X 0,Y 358.875,Z 338.913,A -85,B 0,C 180,E1 -13393.01,E2 -13393.01} C_VEL
LIN {X 0,Y 359.485,Z 345.983,A -85,B 0,C 180,E1 -13393.183,E2 -13393.183} C_VEL
LIN {X 0,Y 358.913,Z 389.137,A -85,B 0,C 180,E1 -13394.069,E2 -13394.069} C_VEL
LIN {X 0,Y 358.461,Z 398.611,A -85,B 0,C 180,E1 -13394.398,E2 -13394.398} C_VEL
LIN {X 0,Y 357.884,Z 408.641,A -85,B 0,C 180,E1 -13394.919,E2 -13394.919} C_VEL
LIN {X 0,Y 357.075,Z 420.046,A -85,B 0,C 180,E1 -13395.758,E2 -13395.758} C_VEL
LIN {X 0,Y 356.315,Z 428.643,A -85,B 0,C 180,E1 -13396.6,E2 -13396.6} C_VEL
LIN {X 0,Y 355.578,Z 436.739,A -85,B 0,C 180,E1 -13397.588,E2 -13397.588} C_VEL
LIN {X 0,Y 355.002,Z 443.435,A -85,B 0,C 180,E1 -13398.582,E2 -13398.582} C_VEL
LIN {X 0,Y 354.433,Z 449.795,A -85,B 0,C 180,E1 -13399.721,E2 -13399.721} C_VEL
LIN {X 0,Y 354.006,Z 455.086,A -85,B 0,C 180,E1 -13400.862,E2 -13400.862} C_VEL
LIN {X 0,Y 353.73,Z 459.504,A -85,B 0,C 180,E1 -13402.006,E2 -13402.006} C_VEL
LIN {X 0,Y 353.453,Z 464.217,A -85,B 0,C 180,E1 -13403.535,E2 -13403.535} C_VEL
LIN {X 0,Y 353.341,Z 467.385,A -85,B 0,C 180,E1 -13404.865,E2 -13404.865} C_VEL
LIN {X 0,Y 353.298,Z 470.316,A -85,B 0,C 180,E1 -13406.579,E2 -13406.579} C_VEL
LIN {X 0,Y 353.343,Z 471.583,A -85,B 0,C 180,E1 -13407.721,E2 -13407.721} C_VEL
LIN {X 0,Y 353.435,Z 472.373,A -85,B 0,C 180,E1 -13408.861,E2 -13408.861} C_VEL
LIN {X 0,Y 353.45,Z 472.67,A -85,B 0,C 180,E1 -13410.001,E2 -13410.001} C_VEL
LIN {X 0,Y 353.435,Z 472.369,A -85,B 0,C 180,E1 -13411.14,E2 -13411.14} C_VEL
LIN {X 0,Y 353.344,Z 471.57,A -85,B 0,C 180,E1 -13412.28,E2 -13412.28} C_VEL
LIN {X 0,Y 353.298,Z 470.295,A -85,B 0,C 180,E1 -13413.422,E2 -13413.422} C_VEL
LIN {X 0,Y 353.341,Z 467.356,A -85,B 0,C 180,E1 -13415.136,E2 -13415.136} C_VEL
LIN {X 0,Y 353.454,Z 464.178,A -85,B 0,C 180,E1 -13416.466,E2 -13416.466} C_VEL
LIN {X 0,Y 353.768,Z 458.482,A -85,B 0,C 180,E1 -13418.282,E2 -13418.282} C_VEL
LIN {X 0,Y 354.175,Z 452.569,A -85,B 0,C 180,E1 -13419.711,E2 -13419.711} C_VEL
LIN {X 0,Y 354.889,Z 445.065,A -85,B 0,C 180,E1 -13421.133,E2 -13421.133} C_VEL
LIN {X 0,Y 355.505,Z 437.665,A -85,B 0,C 180,E1 -13422.27,E2 -13422.27} C_VEL
LIN {X 0,Y 356.204,Z 429.75,A -85,B 0,C 180,E1 -13423.26,E2 -13423.26} C_VEL
LIN {X 0,Y 356.995,Z 421.395,A -85,B 0,C 180,E1 -13424.101,E2 -13424.101} C_VEL
LIN {X 0,Y 357.707,Z 410.714,A -85,B 0,C 180,E1 -13424.944,E2 -13424.944} C_VEL
LIN {X 0,Y 358.39,Z 399.086,A -85,B 0,C 180,E1 -13425.57,E2 -13425.57} C_VEL
LIN {X 0,Y 358.858,Z 389.337,A -85,B 0,C 180,E1 -13425.914,E2 -13425.914} C_VEL
LIN {X 0,Y 359.443,Z 344.351,A -85,B 0,C 180,E1 -13426.838,E2 -13426.838} C_VEL
LIN {X 0,Y 356.275,Z 318.328,A -85,B 0,C 180,E1 -13427.525,E2 -13427.525} C_VEL
LIN {X 0,Y 355.24,Z 311.139,A -85,B 0,C 180,E1 -13427.754,E2 -13427.754} C_VEL
LIN {X 0,Y 356.3,Z 297.508,A -85,B 0,C 180,E1 -13431.099,E2 -13431.099} C_VEL
LIN {X 0,Y 357.278,Z 285.442,A -85,B 0,C 180,E1 -13434.091,E2 -13434.091} C_VEL
LIN {X 0,Y 356.411,Z 279.306,A -85,B 0,C 180,E1 -13435.71,E2 -13435.71} C_VEL
LIN {X 0,Y 354.822,Z 271.099,A -85,B 0,C 180,E1 -13437.981,E2 -13437.981} C_VEL
LIN {X 0,Y 354.776,Z 271.104,A -85,B 0,C 180,E1 -13441.591,E2 -13441.591} C_VEL
LIN {X 0,Y 354.808,Z 271.103,A -85,B 0,C 180,E1 -13445.06,E2 -13445.06} C_VEL
LIN {X 0,Y 354.792,Z 271.1,A -85,B 0,C 180,E1 -13447.885,E2 -13447.885} C_VEL
LIN {X 0,Y 354.767,Z 271.107,A -85,B 0,C 180,E1 -13451.168,E2 -13451.168} C_VEL
LIN {X 0,Y 354.759,Z 271.107,A -85,B 0,C 180,E1 -13454.506,E2 -13454.506} C_VEL
LIN {X 0,Y 354.782,Z 271.101,A -85,B 0,C 180,E1 -13457.661,E2 -13457.661} C_VEL
LIN {X 0,Y 354.786,Z 271.107,A -85,B 0,C 180,E1 -13460.662,E2 -13460.662} C_VEL
LIN {X 0,Y 354.818,Z 271.1,A -85,B 0,C 180,E1 -13464.302,E2 -13464.302} C_VEL
LIN {X 0,Y 354.786,Z 271.101,A -85,B 0,C 180,E1 -13467.667,E2 -13467.667} C_VEL
LIN {X 0,Y 354.789,Z 271.101,A -85,B 0,C 180,E1 -13471.614,E2 -13471.614} C_VEL
LIN {X 0,Y 354.802,Z 271.099,A -85,B 0,C 180,E1 -13475.42,E2 -13475.42} C_VEL
LIN {X 0,Y 354.819,Z 271.097,A -85,B 0,C 180,E1 -13479.113,E2 -13479.113} C_VEL
LIN {X 0,Y 354.837,Z 271.095,A -85,B 0,C 180,E1 -13482.717,E2 -13482.717} C_VEL
LIN {X 0,Y 354.909,Z 271.088,A -85,B 0,C 180,E1 -13486.254,E2 -13486.254} C_VEL
LIN {X 0,Y 354.95,Z 271.086,A -85,B 0,C 180,E1 -13489.735,E2 -13489.735} C_VEL
LIN {X 0,Y 355.088,Z 271.065,A -85,B 0,C 180,E1 -13493.18,E2 -13493.18} C_VEL
LIN {X 0,Y 355.221,Z 271.05,A -85,B 0,C 180,E1 -13497.732,E2 -13497.732} C_VEL
LIN {X 0,Y 355.146,Z 271.059,A -85,B 0,C 180,E1 -13501.134,E2 -13501.134} C_VEL
LIN {X 0,Y 355.226,Z 271.046,A -85,B 0,C 180,E1 -13502.268,E2 -13502.268} C_VEL
LIN {X 0,Y 355.086,Z 271.065,A -85,B 0,C 180,E1 -13506.82,E2 -13506.82} C_VEL
LIN {X 0,Y 354.952,Z 271.08,A -85,B 0,C 180,E1 -13510.265,E2 -13510.265} C_VEL
LIN {X 0,Y 354.925,Z 271.083,A -85,B 0,C 180,E1 -13514.005,E2 -13514.005} C_VEL
LIN {X 0,Y 354.843,Z 271.094,A -85,B 0,C 180,E1 -13518.068,E2 -13518.068} C_VEL
LIN {X 0,Y 354.807,Z 271.099,A -85,B 0,C 180,E1 -13522.108,E2 -13522.108} C_VEL
LIN {X 0,Y 354.801,Z 271.099,A -85,B 0,C 180,E1 -13525.835,E2 -13525.835} C_VEL
LIN {X 0,Y 354.795,Z 271.1,A -85,B 0,C 180,E1 -13529.684,E2 -13529.684} C_VEL
LIN {X 0,Y 354.786,Z 271.105,A -85,B 0,C 180,E1 -13532.334,E2 -13532.334} C_VEL
LIN {X 0,Y 354.82,Z 271.097,A -85,B 0,C 180,E1 -13535.698,E2 -13535.698} C_VEL
LIN {X 0,Y 354.77,Z 271.103,A -85,B 0,C 180,E1 -13539.412,E2 -13539.412} C_VEL
LIN {X 0,Y 354.782,Z 271.102,A -85,B 0,C 180,E1 -13542.866,E2 -13542.866} C_VEL
LIN {X 0,Y 354.764,Z 271.109,A -85,B 0,C 180,E1 -13546.103,E2 -13546.103} C_VEL
LIN {X 0,Y 354.764,Z 271.104,A -85,B 0,C 180,E1 -13549.175,E2 -13549.175} C_VEL
LIN {X 0,Y 354.801,Z 271.1,A -85,B 0,C 180,E1 -13552.404,E2 -13552.404} C_VEL
LIN {X 0,Y 354.81,Z 271.098,A -85,B 0,C 180,E1 -13554.94,E2 -13554.94} C_VEL
LIN {X 0,Y 354.778,Z 271.102,A -85,B 0,C 180,E1 -13558.41,E2 -13558.41} C_VEL
LIN {X 0,Y 354.798,Z 271.105,A -85,B 0,C 180,E1 -13561.614,E2 -13561.614} C_VEL
LIN {X 0,Y 354.842,Z 271.099,A -85,B 0,C 180,E1 -13565.422,E2 -13565.422} C_VEL
LIN {X 0,Y 354.827,Z 271.099,A -85,B 0,C 180,E1 -13569.113,E2 -13569.113} C_VEL
LIN {X 0,Y 354.834,Z 271.103,A -85,B 0,C 180,E1 -13571.374,E2 -13571.374} C_VEL
LIN {X 0,Y 355.458,Z 274.372,A -85,B 0,C 180,E1 -13572.341,E2 -13572.341} C_VEL
LIN {X 0,Y 358.134,Z 283.509,A -85,B 0,C 180,E1 -13572.672,E2 -13572.672} C_VEL
LIN {X 0,Y 360.092,Z 293.492,A -85,B 0,C 180,E1 -13572.976,E2 -13572.976} C_VEL
LIN {X 0,Y 359.241,Z 349.601,A -85,B 0,C 180,E1 -13574.104,E2 -13574.104} C_VEL
LIN {X 0,Y 359.083,Z 359.066,A -85,B 0,C 180,E1 -13574.424,E2 -13574.424} C_VEL
LIN {X 0,Y 358.824,Z 368.221,A -85,B 0,C 180,E1 -13574.885,E2 -13574.885} C_VEL
LIN {X 0,Y 358.363,Z 377.558,A -85,B 0,C 180,E1 -13575.519,E2 -13575.519} C_VEL
LIN {X 0,Y 357.657,Z 387.124,A -85,B 0,C 180,E1 -13576.361,E2 -13576.361} C_VEL
LIN {X 0,Y 357.011,Z 396.883,A -85,B 0,C 180,E1 -13577.493,E2 -13577.493} C_VEL
LIN {X 0,Y 356.3,Z 404.588,A -85,B 0,C 180,E1 -13578.623,E2 -13578.623} C_VEL
LIN {X 0,Y 355.664,Z 410.92,A -85,B 0,C 180,E1 -13579.755,E2 -13579.755} C_VEL
LIN {X 0,Y 355.017,Z 417.343,A -85,B 0,C 180,E1 -13581.174,E2 -13581.174} C_VEL
LIN {X 0,Y 354.57,Z 422.664,A -85,B 0,C 180,E1 -13582.658,E2 -13582.658} C_VEL
LIN {X 0,Y 354.062,Z 427.203,A -85,B 0,C 180,E1 -13584.304,E2 -13584.304} C_VEL
LIN {X 0,Y 353.89,Z 429.508,A -85,B 0,C 180,E1 -13585.443,E2 -13585.443} C_VEL
LIN {X 0,Y 353.783,Z 431.261,A -85,B 0,C 180,E1 -13586.583,E2 -13586.583} C_VEL
LIN {X 0,Y 353.623,Z 432.53,A -85,B 0,C 180,E1 -13587.721,E2 -13587.721} C_VEL
LIN {X 0,Y 353.494,Z 433.333,A -85,B 0,C 180,E1 -13588.86,E2 -13588.86} C_VEL
LIN {X 0,Y 353.457,Z 433.639,A -85,B 0,C 180,E1 -13589.999,E2 -13589.999} C_VEL
LIN {X 0,Y 353.494,Z 433.362,A -85,B 0,C 180,E1 -13591.139,E2 -13591.139} C_VEL
LIN {X 0,Y 353.602,Z 432.62,A -85,B 0,C 180,E1 -13592.278,E2 -13592.278} C_VEL
LIN {X 0,Y 353.778,Z 431.41,A -85,B 0,C 180,E1 -13593.416,E2 -13593.416} C_VEL
LIN {X 0,Y 353.963,Z 428.581,A -85,B 0,C 180,E1 -13595.125,E2 -13595.125} C_VEL
LIN {X 0,Y 354.205,Z 426.001,A -85,B 0,C 180,E1 -13596.264,E2 -13596.264} C_VEL
LIN {X 0,Y 354.723,Z 421.324,A -85,B 0,C 180,E1 -13597.848,E2 -13597.848} C_VEL
LIN {X 0,Y 355.104,Z 416.613,A -85,B 0,C 180,E1 -13599.109,E2 -13599.109} C_VEL
LIN {X 0,Y 355.601,Z 411.441,A -85,B 0,C 180,E1 -13600.245,E2 -13600.245} C_VEL
LIN {X 0,Y 356.286,Z 405.203,A -85,B 0,C 180,E1 -13601.376,E2 -13601.376} C_VEL
LIN {X 0,Y 356.961,Z 397.622,A -85,B 0,C 180,E1 -13602.507,E2 -13602.507} C_VEL
LIN {X 0,Y 357.651,Z 388.179,A -85,B 0,C 180,E1 -13603.638,E2 -13603.638} C_VEL
LIN {X 0,Y 358.313,Z 378.92,A -85,B 0,C 180,E1 -13604.482,E2 -13604.482} C_VEL
LIN {X 0,Y 358.799,Z 369.978,A -85,B 0,C 180,E1 -13605.114,E2 -13605.114} C_VEL
LIN {X 0,Y 359.101,Z 360.652,A -85,B 0,C 180,E1 -13605.61,E2 -13605.61} C_VEL
LIN {X 0,Y 359.298,Z 351.182,A -85,B 0,C 180,E1 -13605.954,E2 -13605.954} C_VEL
LIN {X 0,Y 360.07,Z 293.286,A -85,B 0,C 180,E1 -13607.134,E2 -13607.134} C_VEL
LIN {X 0,Y 357.169,Z 279.757,A -85,B 0,C 180,E1 -13607.561,E2 -13607.561} C_VEL
LIN {X 0,Y 355.428,Z 274.264,A -85,B 0,C 180,E1 -13607.798,E2 -13607.798} C_VEL
LIN {X 0,Y 355.217,Z 273.11,A -85,B 0,C 180,E1 -13608.138,E2 -13608.138} C_VEL
LIN {X 0,Y 354.568,Z 271.797,A -85,B 0,C 180,E1 -13608.711,E2 -13608.711} C_VEL
LIN {X 0,Y 353.557,Z 271.305,A -85,B 0,C 180,E1 -13609.31,E2 -13609.31} C_VEL
LIN {X 0,Y 348.762,Z 271.902,A -85,B 0,C 180,E1 -13611.817,E2 -13611.817} C_VEL
LIN {X 0,Y 347.807,Z 271.977,A -85,B 0,C 180,E1 -13612.807,E2 -13612.807} C_VEL
LIN {X 0,Y 347.731,Z 271.98,A -85,B 0,C 180,E1 -13613.141,E2 -13613.141} C_VEL
LIN {X 0,Y 347.733,Z 271.984,A -85,B 0,C 180,E1 -13616.399,E2 -13616.399} C_VEL
LIN {X 0,Y 347.727,Z 271.985,A -85,B 0,C 180,E1 -13620.349,E2 -13620.349} C_VEL
LIN {X 0,Y 347.746,Z 271.981,A -85,B 0,C 180,E1 -13624.043,E2 -13624.043} C_VEL
LIN {X 0,Y 347.753,Z 271.977,A -85,B 0,C 180,E1 -13627.321,E2 -13627.321} C_VEL
LIN {X 0,Y 347.692,Z 271.988,A -85,B 0,C 180,E1 -13630.302,E2 -13630.302} C_VEL
LIN {X 0,Y 347.717,Z 271.982,A -85,B 0,C 180,E1 -13633.408,E2 -13633.408} C_VEL
LIN {X 0,Y 347.719,Z 271.981,A -85,B 0,C 180,E1 -13636.686,E2 -13636.686} C_VEL
LIN {X 0,Y 347.697,Z 271.986,A -85,B 0,C 180,E1 -13640.182,E2 -13640.182} C_VEL
LIN {X 0,Y 347.751,Z 271.977,A -85,B 0,C 180,E1 -13642.678,E2 -13642.678} C_VEL
LIN {X 0,Y 347.744,Z 271.981,A -85,B 0,C 180,E1 -13645.956,E2 -13645.956} C_VEL
LIN {X 0,Y 347.731,Z 271.984,A -85,B 0,C 180,E1 -13649.65,E2 -13649.65} C_VEL
LIN {X 0,Y 347.734,Z 271.983,A -85,B 0,C 180,E1 -13653.6,E2 -13653.6} C_VEL
LIN {X 0,Y 347.754,Z 271.977,A -85,B 0,C 180,E1 -13656.159,E2 -13656.159} C_VEL
LIN {X 0,Y 347.766,Z 271.976,A -85,B 0,C 180,E1 -13659.906,E2 -13659.906} C_VEL
LIN {X 0,Y 347.792,Z 271.973,A -85,B 0,C 180,E1 -13663.566,E2 -13663.566} C_VEL
LIN {X 0,Y 347.879,Z 271.965,A -85,B 0,C 180,E1 -13667.16,E2 -13667.16} C_VEL
LIN {X 0,Y 347.928,Z 271.959,A -85,B 0,C 180,E1 -13670.7,E2 -13670.7} C_VEL
LIN {X 0,Y 348.031,Z 271.943,A -85,B 0,C 180,E1 -13674.205,E2 -13674.205} C_VEL
LIN {X 0,Y 348.181,Z 271.923,A -85,B 0,C 180,E1 -13677.686,E2 -13677.686} C_VEL
LIN {X 0,Y 348.11,Z 271.933,A -85,B 0,C 180,E1 -13681.157,E2 -13681.157} C_VEL
LIN {X 0,Y 348.181,Z 271.927,A -85,B 0,C 180,E1 -13682.314,E2 -13682.314} C_VEL
LIN {X 0,Y 348.046,Z 271.941,A -85,B 0,C 180,E1 -13686.959,E2 -13686.959} C_VEL
LIN {X 0,Y 347.885,Z 271.964,A -85,B 0,C 180,E1 -13690.476,E2 -13690.476} C_VEL
LIN {X 0,Y 347.874,Z 271.967,A -85,B 0,C 180,E1 -13694.137,E2 -13694.137} C_VEL
LIN {X 0,Y 347.787,Z 271.976,A -85,B 0,C 180,E1 -13698.241,E2 -13698.241} C_VEL
LIN {X 0,Y 347.757,Z 271.979,A -85,B 0,C 180,E1 -13701.624,E2 -13701.624} C_VEL
LIN {X 0,Y 347.728,Z 271.98,A -85,B 0,C 180,E1 -13705.115,E2 -13705.115} C_VEL
LIN {X 0,Y 347.72,Z 271.987,A -85,B 0,C 180,E1 -13707.702,E2 -13707.702} C_VEL
LIN {X 0,Y 347.73,Z 271.98,A -85,B 0,C 180,E1 -13710.35,E2 -13710.35} C_VEL
LIN {X 0,Y 347.744,Z 271.979,A -85,B 0,C 180,E1 -13714.044,E2 -13714.044} C_VEL
LIN {X 0,Y 347.75,Z 271.982,A -85,B 0,C 180,E1 -13717.322,E2 -13717.322} C_VEL
LIN {X 0,Y 347.691,Z 271.984,A -85,B 0,C 180,E1 -13720.303,E2 -13720.303} C_VEL
LIN {X 0,Y 347.716,Z 271.986,A -85,B 0,C 180,E1 -13723.409,E2 -13723.409} C_VEL
LIN {X 0,Y 347.718,Z 271.983,A -85,B 0,C 180,E1 -13726.687,E2 -13726.687} C_VEL
LIN {X 0,Y 347.696,Z 271.984,A -85,B 0,C 180,E1 -13730.183,E2 -13730.183} C_VEL
LIN {X 0,Y 347.75,Z 271.98,A -85,B 0,C 180,E1 -13732.679,E2 -13732.679} C_VEL
LIN {X 0,Y 347.745,Z 271.978,A -85,B 0,C 180,E1 -13735.957,E2 -13735.957} C_VEL
LIN {X 0,Y 347.726,Z 271.98,A -85,B 0,C 180,E1 -13739.651,E2 -13739.651} C_VEL
LIN {X 0,Y 347.79,Z 272.15,A -85,B 0,C 180,E1 -13741.814,E2 -13741.814} C_VEL
LIN {X 0,Y 349.819,Z 282.526,A -85,B 0,C 180,E1 -13744.698,E2 -13744.698} C_VEL
LIN {X 0,Y 350.293,Z 286.319,A -85,B 0,C 180,E1 -13745.715,E2 -13745.715} C_VEL
LIN {X 0,Y 349.214,Z 299.586,A -85,B 0,C 180,E1 -13749.071,E2 -13749.071} C_VEL
LIN {X 0,Y 348.323,Z 311.037,A -85,B 0,C 180,E1 -13751.901,E2 -13751.901} C_VEL
LIN {X 0,Y 351.924,Z 337.969,A -85,B 0,C 180,E1 -13752.652,E2 -13752.652} C_VEL
LIN {X 0,Y 352.686,Z 347.071,A -85,B 0,C 180,E1 -13752.879,E2 -13752.879} C_VEL
LIN {X 0,Y 352.1,Z 388.12,A -85,B 0,C 180,E1 -13753.734,E2 -13753.734} C_VEL
LIN {X 0,Y 351.672,Z 397.396,A -85,B 0,C 180,E1 -13754.051,E2 -13754.051} C_VEL
LIN {X 0,Y 351.103,Z 407.044,A -85,B 0,C 180,E1 -13754.546,E2 -13754.546} C_VEL
LIN {X 0,Y 350.442,Z 416.205,A -85,B 0,C 180,E1 -13755.186,E2 -13755.186} C_VEL
LIN {X 0,Y 349.546,Z 427.019,A -85,B 0,C 180,E1 -13756.187,E2 -13756.187} C_VEL
LIN {X 0,Y 348.64,Z 436.349,A -85,B 0,C 180,E1 -13757.337,E2 -13757.337} C_VEL
LIN {X 0,Y 348.015,Z 443.044,A -85,B 0,C 180,E1 -13758.35,E2 -13758.35} C_VEL
LIN {X 0,Y 347.428,Z 449.404,A -85,B 0,C 180,E1 -13759.511,E2 -13759.511} C_VEL
LIN {X 0,Y 346.977,Z 454.694,A -85,B 0,C 180,E1 -13760.675,E2 -13760.675} C_VEL
LIN {X 0,Y 346.668,Z 459.112,A -85,B 0,C 180,E1 -13761.842,E2 -13761.842} C_VEL
LIN {X 0,Y 346.348,Z 464.479,A -85,B 0,C 180,E1 -13763.651,E2 -13763.651} C_VEL
LIN {X 0,Y 346.271,Z 468.162,A -85,B 0,C 180,E1 -13765.344,E2 -13765.344} C_VEL
LIN {X 0,Y 346.219,Z 469.925,A -85,B 0,C 180,E1 -13766.509,E2 -13766.509} C_VEL
LIN {X 0,Y 346.246,Z 471.191,A -85,B 0,C 180,E1 -13767.674,E2 -13767.674} C_VEL
LIN {X 0,Y 346.353,Z 471.982,A -85,B 0,C 180,E1 -13768.838,E2 -13768.838} C_VEL
LIN {X 0,Y 346.387,Z 472.28,A -85,B 0,C 180,E1 -13770.001,E2 -13770.001} C_VEL
LIN {X 0,Y 346.353,Z 471.978,A -85,B 0,C 180,E1 -13771.163,E2 -13771.163} C_VEL
LIN {X 0,Y 346.246,Z 471.177,A -85,B 0,C 180,E1 -13772.327,E2 -13772.327} C_VEL
LIN {X 0,Y 346.219,Z 469.903,A -85,B 0,C 180,E1 -13773.492,E2 -13773.492} C_VEL
LIN {X 0,Y 346.239,Z 466.961,A -85,B 0,C 180,E1 -13775.241,E2 -13775.241} C_VEL
LIN {X 0,Y 346.349,Z 464.438,A -85,B 0,C 180,E1 -13776.35,E2 -13776.35} C_VEL
LIN {X 0,Y 346.655,Z 459.057,A -85,B 0,C 180,E1 -13778.159,E2 -13778.159} C_VEL
LIN {X 0,Y 347.155,Z 452.173,A -85,B 0,C 180,E1 -13779.909,E2 -13779.909} C_VEL
LIN {X 0,Y 347.878,Z 444.668,A -85,B 0,C 180,E1 -13781.361,E2 -13781.361} C_VEL
LIN {X 0,Y 348.533,Z 437.268,A -85,B 0,C 180,E1 -13782.52,E2 -13782.52} C_VEL
LIN {X 0,Y 349.291,Z 429.354,A -85,B 0,C 180,E1 -13783.528,E2 -13783.528} C_VEL
LIN {X 0,Y 350.105,Z 420.998,A -85,B 0,C 180,E1 -13784.384,E2 -13784.384} C_VEL
LIN {X 0,Y 350.855,Z 410.316,A -85,B 0,C 180,E1 -13785.243,E2 -13785.243} C_VEL
LIN {X 0,Y 351.57,Z 398.685,A -85,B 0,C 180,E1 -13785.88,E2 -13785.88} C_VEL
LIN {X 0,Y 352.039,Z 388.93,A -85,B 0,C 180,E1 -13786.23,E2 -13786.23} C_VEL
LIN {X 0,Y 352.669,Z 345.287,A -85,B 0,C 180,E1 -13787.143,E2 -13787.143} C_VEL
LIN {X 0,Y 349.457,Z 318.93,A -85,B 0,C 180,E1 -13787.857,E2 -13787.857} C_VEL
LIN {X 0,Y 348.272,Z 310.847,A -85,B 0,C 180,E1 -13788.094,E2 -13788.094} C_VEL
LIN {X 0,Y 349.38,Z 297.13,A -85,B 0,C 180,E1 -13791.532,E2 -13791.532} C_VEL
LIN {X 0,Y 350.296,Z 286.245,A -85,B 0,C 180,E1 -13794.287,E2 -13794.287} C_VEL
LIN {X 0,Y 348.947,Z 277.718,A -85,B 0,C 180,E1 -13796.604,E2 -13796.604} C_VEL
LIN {X 0,Y 347.775,Z 271.976,A -85,B 0,C 180,E1 -13798.271,E2 -13798.271} C_VEL
LIN {X 0,Y 347.726,Z 271.98,A -85,B 0,C 180,E1 -13801.911,E2 -13801.911} C_VEL
LIN {X 0,Y 347.784,Z 271.973,A -85,B 0,C 180,E1 -13805.876,E2 -13805.876} C_VEL
LIN {X 0,Y 347.731,Z 271.983,A -85,B 0,C 180,E1 -13808.796,E2 -13808.796} C_VEL
LIN {X 0,Y 347.74,Z 271.978,A -85,B 0,C 180,E1 -13811.832,E2 -13811.832} C_VEL
LIN {X 0,Y 347.701,Z 271.987,A -85,B 0,C 180,E1 -13815.028,E2 -13815.028} C_VEL
LIN {X 0,Y 347.738,Z 271.981,A -85,B 0,C 180,E1 -13818.4,E2 -13818.4} C_VEL
LIN {X 0,Y 347.762,Z 271.977,A -85,B 0,C 180,E1 -13822.014,E2 -13822.014} C_VEL
LIN {X 0,Y 347.743,Z 271.978,A -85,B 0,C 180,E1 -13825.536,E2 -13825.536} C_VEL
LIN {X 0,Y 347.745,Z 271.983,A -85,B 0,C 180,E1 -13828.301,E2 -13828.301} C_VEL
LIN {X 0,Y 347.741,Z 271.979,A -85,B 0,C 180,E1 -13830.984,E2 -13830.984} C_VEL
LIN {X 0,Y 347.732,Z 271.98,A -85,B 0,C 180,E1 -13833.6,E2 -13833.6} C_VEL
LIN {X 0,Y 347.748,Z 271.983,A -85,B 0,C 180,E1 -13836.159,E2 -13836.159} C_VEL
LIN {X 0,Y 347.764,Z 271.98,A -85,B 0,C 180,E1 -13839.907,E2 -13839.907} C_VEL
LIN {X 0,Y 347.783,Z 271.975,A -85,B 0,C 180,E1 -13843.566,E2 -13843.566} C_VEL
LIN {X 0,Y 347.864,Z 271.963,A -85,B 0,C 180,E1 -13847.16,E2 -13847.16} C_VEL
LIN {X 0,Y 347.935,Z 271.954,A -85,B 0,C 180,E1 -13850.701,E2 -13850.701} C_VEL
LIN {X 0,Y 348.037,Z 271.942,A -85,B 0,C 180,E1 -13854.205,E2 -13854.205} C_VEL
LIN {X 0,Y 348.182,Z 271.928,A -85,B 0,C 180,E1 -13857.686,E2 -13857.686} C_VEL
LIN {X 0,Y 348.118,Z 271.935,A -85,B 0,C 180,E1 -13861.157,E2 -13861.157} C_VEL
LIN {X 0,Y 348.188,Z 271.922,A -85,B 0,C 180,E1 -13862.314,E2 -13862.314} C_VEL
LIN {X 0,Y 348.054,Z 271.942,A -85,B 0,C 180,E1 -13866.959,E2 -13866.959} C_VEL
LIN {X 0,Y 347.893,Z 271.96,A -85,B 0,C 180,E1 -13870.476,E2 -13870.476} C_VEL
LIN {X 0,Y 347.882,Z 271.96,A -85,B 0,C 180,E1 -13874.137,E2 -13874.137} C_VEL
LIN {X 0,Y 347.794,Z 271.972,A -85,B 0,C 180,E1 -13878.241,E2 -13878.241} C_VEL
LIN {X 0,Y 347.765,Z 271.975,A -85,B 0,C 180,E1 -13881.624,E2 -13881.624} C_VEL
LIN {X 0,Y 347.738,Z 271.98,A -85,B 0,C 180,E1 -13885.114,E2 -13885.114} C_VEL
LIN {X 0,Y 347.73,Z 271.979,A -85,B 0,C 180,E1 -13887.701,E2 -13887.701} C_VEL
LIN {X 0,Y 347.737,Z 271.983,A -85,B 0,C 180,E1 -13890.349,E2 -13890.349} C_VEL
LIN {X 0,Y 347.75,Z 271.979,A -85,B 0,C 180,E1 -13894.043,E2 -13894.043} C_VEL
LIN {X 0,Y 347.757,Z 271.976,A -85,B 0,C 180,E1 -13897.322,E2 -13897.322} C_VEL
LIN {X 0,Y 347.697,Z 271.989,A -85,B 0,C 180,E1 -13900.302,E2 -13900.302} C_VEL
LIN {X 0,Y 347.722,Z 271.981,A -85,B 0,C 180,E1 -13903.408,E2 -13903.408} C_VEL
LIN {X 0,Y 347.724,Z 271.981,A -85,B 0,C 180,E1 -13906.687,E2 -13906.687} C_VEL
LIN {X 0,Y 347.702,Z 271.986,A -85,B 0,C 180,E1 -13910.182,E2 -13910.182} C_VEL
LIN {X 0,Y 347.757,Z 271.976,A -85,B 0,C 180,E1 -13912.678,E2 -13912.678} C_VEL
LIN {X 0,Y 347.75,Z 271.981,A -85,B 0,C 180,E1 -13915.956,E2 -13915.956} C_VEL
LIN {X 0,Y 347.731,Z 271.986,A -85,B 0,C 180,E1 -13919.65,E2 -13919.65} C_VEL
LIN {X 0,Y 347.741,Z 271.984,A -85,B 0,C 180,E1 -13923.6,E2 -13923.6} C_VEL
LIN {X 0,Y 347.761,Z 271.976,A -85,B 0,C 180,E1 -13926.159,E2 -13926.159} C_VEL
LIN {X 0,Y 347.779,Z 271.98,A -85,B 0,C 180,E1 -13929.907,E2 -13929.907} C_VEL
LIN {X 0,Y 347.829,Z 272.018,A -85,B 0,C 180,E1 -13931.138,E2 -13931.138} C_VEL
LIN {X 0,Y 348.347,Z 274.772,A -85,B 0,C 180,E1 -13931.968,E2 -13931.968} C_VEL
LIN {X 0,Y 351.628,Z 285.725,A -85,B 0,C 180,E1 -13932.379,E2 -13932.379} C_VEL
LIN {X 0,Y 353.341,Z 295.146,A -85,B 0,C 180,E1 -13932.667,E2 -13932.667} C_VEL
LIN {X 0,Y 352.463,Z 351.302,A -85,B 0,C 180,E1 -13933.827,E2 -13933.827} C_VEL
LIN {X 0,Y 352.262,Z 360.296,A -85,B 0,C 180,E1 -13934.152,E2 -13934.152} C_VEL
LIN {X 0,Y 351.948,Z 369.826,A -85,B 0,C 180,E1 -13934.657,E2 -13934.657} C_VEL
LIN {X 0,Y 351.38,Z 379.822,A -85,B 0,C 180,E1 -13935.373,E2 -13935.373} C_VEL
LIN {X 0,Y 350.67,Z 390.183,A -85,B 0,C 180,E1 -13936.379,E2 -13936.379} C_VEL
LIN {X 0,Y 349.993,Z 398.293,A -85,B 0,C 180,E1 -13937.386,E2 -13937.386} C_VEL
LIN {X 0,Y 349.362,Z 404.982,A -85,B 0,C 180,E1 -13938.394,E2 -13938.394} C_VEL
LIN {X 0,Y 348.704,Z 411.313,A -85,B 0,C 180,E1 -13939.549,E2 -13939.549} C_VEL
LIN {X 0,Y 348.036,Z 417.735,A -85,B 0,C 180,E1 -13940.996,E2 -13940.996} C_VEL
LIN {X 0,Y 347.69,Z 421.65,A -85,B 0,C 180,E1 -13942.079,E2 -13942.079} C_VEL
LIN {X 0,Y 347.197,Z 426.114,A -85,B 0,C 180,E1 -13943.607,E2 -13943.607} C_VEL
LIN {X 0,Y 346.915,Z 428.762,A -85,B 0,C 180,E1 -13944.769,E2 -13944.769} C_VEL
LIN {X 0,Y 346.702,Z 431.654,A -85,B 0,C 180,E1 -13946.513,E2 -13946.513} C_VEL
LIN {X 0,Y 346.55,Z 432.921,A -85,B 0,C 180,E1 -13947.675,E2 -13947.675} C_VEL
LIN {X 0,Y 346.434,Z 433.723,A -85,B 0,C 180,E1 -13948.837,E2 -13948.837} C_VEL
LIN {X 0,Y 346.394,Z 434.029,A -85,B 0,C 180,E1 -13949.999,E2 -13949.999} C_VEL
LIN {X 0,Y 346.433,Z 433.752,A -85,B 0,C 180,E1 -13951.162,E2 -13951.162} C_VEL
LIN {X 0,Y 346.531,Z 433.01,A -85,B 0,C 180,E1 -13952.324,E2 -13952.324} C_VEL
LIN {X 0,Y 346.697,Z 431.801,A -85,B 0,C 180,E1 -13953.486,E2 -13953.486} C_VEL
LIN {X 0,Y 346.899,Z 428.971,A -85,B 0,C 180,E1 -13955.23,E2 -13955.23} C_VEL
LIN {X 0,Y 347.18,Z 426.39,A -85,B 0,C 180,E1 -13956.392,E2 -13956.392} C_VEL
LIN {X 0,Y 347.674,Z 422.056,A -85,B 0,C 180,E1 -13957.902,E2 -13957.902} C_VEL
LIN {X 0,Y 348.108,Z 417.002,A -85,B 0,C 180,E1 -13959.294,E2 -13959.294} C_VEL
LIN {X 0,Y 348.64,Z 411.83,A -85,B 0,C 180,E1 -13960.452,E2 -13960.452} C_VEL
LIN {X 0,Y 349.334,Z 405.592,A -85,B 0,C 180,E1 -13961.605,E2 -13961.605} C_VEL
LIN {X 0,Y 350.055,Z 398.009,A -85,B 0,C 180,E1 -13962.758,E2 -13962.758} C_VEL
LIN {X 0,Y 350.784,Z 388.564,A -85,B 0,C 180,E1 -13963.911,E2 -13963.911} C_VEL
LIN {X 0,Y 351.465,Z 379.305,A -85,B 0,C 180,E1 -13964.77,E2 -13964.77} C_VEL
LIN {X 0,Y 351.985,Z 370.359,A -85,B 0,C 180,E1 -13965.414,E2 -13965.414} C_VEL
LIN {X 0,Y 352.299,Z 361.03,A -85,B 0,C 180,E1 -13965.919,E2 -13965.919} C_VEL
LIN {X 0,Y 352.491,Z 351.648,A -85,B 0,C 180,E1 -13966.268,E2 -13966.268} C_VEL
LIN {X 0,Y 353.311,Z 294.316,A -85,B 0,C 180,E1 -13967.459,E2 -13967.459} C_VEL
LIN {X 0,Y 350.78,Z 282.304,A -85,B 0,C 180,E1 -13967.845,E2 -13967.845} C_VEL
LIN {X 0,Y 348.327,Z 274.753,A -85,B 0,C 180,E1 -13968.148,E2 -13968.148} C_VEL
LIN {X 0,Y 347.802,Z 271.978,A -85,B 0,C 180,E1 -13969.015,E2 -13969.015} C_VEL
LIN {X 0,Y 347.753,Z 271.982,A -85,B 0,C 180,E1 -13972.58,E2 -13972.58} C_VEL
LIN {X 0,Y 347.731,Z 271.98,A -85,B 0,C 180,E1 -13973.141,E2 -13973.141} C_VEL
LIN {X 0,Y 347.059,Z 272.066,A -85,B 0,C 180,E1 -13974.107,E2 -13974.107} C_VEL
LIN {X 0,Y 344.189,Z 272.421,A -85,B 0,C 180,E1 -13975.678,E2 -13975.678} C_VEL
LIN {X 0,Y 341.771,Z 272.724,A -85,B 0,C 180,E1 -13976.95,E2 -13976.95} C_VEL
LIN {X 0,Y 340.749,Z 272.851,A -85,B 0,C 180,E1 -13977.935,E2 -13977.935} C_VEL
LIN {X 0,Y 340.675,Z 272.862,A -85,B 0,C 180,E1 -13978.268,E2 -13978.268} C_VEL
LIN {X 0,Y 340.68,Z 272.859,A -85,B 0,C 180,E1 -13981.046,E2 -13981.046} C_VEL
LIN {X 0,Y 340.713,Z 272.853,A -85,B 0,C 180,E1 -13985.278,E2 -13985.278} C_VEL
LIN {X 0,Y 340.691,Z 272.86,A -85,B 0,C 180,E1 -13988.382,E2 -13988.382} C_VEL
LIN {X 0,Y 340.687,Z 272.862,A -85,B 0,C 180,E1 -13992.043,E2 -13992.043} C_VEL
LIN {X 0,Y 340.646,Z 272.865,A -85,B 0,C 180,E1 -13996.227,E2 -13996.227} C_VEL
LIN {X 0,Y 340.664,Z 272.859,A -85,B 0,C 180,E1 -13998.687,E2 -13998.687} C_VEL
LIN {X 0,Y 340.715,Z 272.859,A -85,B 0,C 180,E1 -14001.77,E2 -14001.77} C_VEL
LIN {X 0,Y 340.718,Z 272.858,A -85,B 0,C 180,E1 -14005.595,E2 -14005.595} C_VEL
LIN {X 0,Y 340.686,Z 272.858,A -85,B 0,C 180,E1 -14008.954,E2 -14008.954} C_VEL
LIN {X 0,Y 340.707,Z 272.856,A -85,B 0,C 180,E1 -14013.011,E2 -14013.011} C_VEL
LIN {X 0,Y 340.74,Z 272.853,A -85,B 0,C 180,E1 -14015.637,E2 -14015.637} C_VEL
LIN {X 0,Y 340.707,Z 272.858,A -85,B 0,C 180,E1 -14019.471,E2 -14019.471} C_VEL
LIN {X 0,Y 340.755,Z 272.848,A -85,B 0,C 180,E1 -14021.978,E2 -14021.978} C_VEL
LIN {X 0,Y 340.827,Z 272.839,A -85,B 0,C 180,E1 -14025.73,E2 -14025.73} C_VEL
LIN {X 0,Y 340.838,Z 272.84,A -85,B 0,C 180,E1 -14029.305,E2 -14029.305} C_VEL
LIN {X 0,Y 340.995,Z 272.823,A -85,B 0,C 180,E1 -14032.896,E2 -14032.896} C_VEL
LIN {X 0,Y 340.803,Z 272.842,A -85,B 0,C 180,E1 -14035.268,E2 -14035.268} C_VEL
LIN {X 0,Y 341.118,Z 272.802,A -85,B 0,C 180,E1 -14037.638,E2 -14037.638} C_VEL
LIN {X 0,Y 341.082,Z 272.809,A -85,B 0,C 180,E1 -14041.181,E2 -14041.181} C_VEL
LIN {X 0,Y 341.118,Z 272.807,A -85,B 0,C 180,E1 -14042.361,E2 -14042.361} C_VEL
LIN {X 0,Y 340.994,Z 272.819,A -85,B 0,C 180,E1 -14047.103,E2 -14047.103} C_VEL
LIN {X 0,Y 340.838,Z 272.84,A -85,B 0,C 180,E1 -14050.695,E2 -14050.695} C_VEL
LIN {X 0,Y 340.813,Z 272.845,A -85,B 0,C 180,E1 -14054.327,E2 -14054.327} C_VEL
LIN {X 0,Y 340.749,Z 272.851,A -85,B 0,C 180,E1 -14058.425,E2 -14058.425} C_VEL
LIN {X 0,Y 340.713,Z 272.859,A -85,B 0,C 180,E1 -14061.842,E2 -14061.842} C_VEL
LIN {X 0,Y 340.699,Z 272.855,A -85,B 0,C 180,E1 -14064.821,E2 -14064.821} C_VEL
LIN {X 0,Y 340.67,Z 272.86,A -85,B 0,C 180,E1 -14068.326,E2 -14068.326} C_VEL
LIN {X 0,Y 340.687,Z 272.858,A -85,B 0,C 180,E1 -14071.046,E2 -14071.046} C_VEL
LIN {X 0,Y 340.712,Z 272.858,A -85,B 0,C 180,E1 -14075.279,E2 -14075.279} C_VEL
LIN {X 0,Y 340.688,Z 272.857,A -85,B 0,C 180,E1 -14078.383,E2 -14078.383} C_VEL
LIN {X 0,Y 340.686,Z 272.858,A -85,B 0,C 180,E1 -14082.044,E2 -14082.044} C_VEL
LIN {X 0,Y 340.645,Z 272.862,A -85,B 0,C 180,E1 -14086.228,E2 -14086.228} C_VEL
LIN {X 0,Y 340.664,Z 272.862,A -85,B 0,C 180,E1 -14088.688,E2 -14088.688} C_VEL
LIN {X 0,Y 340.714,Z 272.854,A -85,B 0,C 180,E1 -14091.771,E2 -14091.771} C_VEL
LIN {X 0,Y 340.718,Z 272.854,A -85,B 0,C 180,E1 -14095.596,E2 -14095.596} C_VEL
LIN {X 0,Y 340.679,Z 272.862,A -85,B 0,C 180,E1 -14098.954,E2 -14098.954} C_VEL
LIN {X 0,Y 340.724,Z 272.95,A -85,B 0,C 180,E1 -14101.512,E2 -14101.512} C_VEL
LIN {X 0,Y 342.804,Z 283.446,A -85,B 0,C 180,E1 -14104.5,E2 -14104.5} C_VEL
LIN {X 0,Y 343.254,Z 288.335,A -85,B 0,C 180,E1 -14105.828,E2 -14105.828} C_VEL
LIN {X 0,Y 342.011,Z 302.792,A -85,B 0,C 180,E1 -14109.554,E2 -14109.554} C_VEL
LIN {X 0,Y 341.366,Z 310.462,A -85,B 0,C 180,E1 -14111.514,E2 -14111.514} C_VEL
LIN {X 0,Y 344.831,Z 336.073,A -85,B 0,C 180,E1 -14112.251,E2 -14112.251} C_VEL
LIN {X 0,Y 345.881,Z 347.634,A -85,B 0,C 180,E1 -14112.552,E2 -14112.552} C_VEL
LIN {X 0,Y 345.272,Z 387.857,A -85,B 0,C 180,E1 -14113.406,E2 -14113.406} C_VEL
LIN {X 0,Y 344.85,Z 397.014,A -85,B 0,C 180,E1 -14113.727,E2 -14113.727} C_VEL
LIN {X 0,Y 344.269,Z 406.659,A -85,B 0,C 180,E1 -14114.231,E2 -14114.231} C_VEL
LIN {X 0,Y 343.572,Z 415.818,A -85,B 0,C 180,E1 -14114.883,E2 -14114.883} C_VEL
LIN {X 0,Y 342.66,Z 426.631,A -85,B 0,C 180,E1 -14115.904,E2 -14115.904} C_VEL
LIN {X 0,Y 341.692,Z 435.959,A -85,B 0,C 180,E1 -14117.075,E2 -14117.075} C_VEL
LIN {X 0,Y 341.032,Z 442.652,A -85,B 0,C 180,E1 -14118.108,E2 -14118.108} C_VEL
LIN {X 0,Y 340.438,Z 449.014,A -85,B 0,C 180,E1 -14119.293,E2 -14119.293} C_VEL
LIN {X 0,Y 339.948,Z 454.303,A -85,B 0,C 180,E1 -14120.481,E2 -14120.481} C_VEL
LIN {X 0,Y 339.613,Z 458.72,A -85,B 0,C 180,E1 -14121.672,E2 -14121.672} C_VEL
LIN {X 0,Y 339.297,Z 463.936,A -85,B 0,C 180,E1 -14123.46,E2 -14123.46} C_VEL
LIN {X 0,Y 339.182,Z 467.77,A -85,B 0,C 180,E1 -14125.246,E2 -14125.246} C_VEL
LIN {X 0,Y 339.142,Z 469.534,A -85,B 0,C 180,E1 -14126.436,E2 -14126.436} C_VEL
LIN {X 0,Y 339.149,Z 470.799,A -85,B 0,C 180,E1 -14127.625,E2 -14127.625} C_VEL
LIN {X 0,Y 339.257,Z 471.59,A -85,B 0,C 180,E1 -14128.814,E2 -14128.814} C_VEL
LIN {X 0,Y 339.325,Z 471.89,A -85,B 0,C 180,E1 -14130.001,E2 -14130.001} C_VEL
LIN {X 0,Y 339.257,Z 471.586,A -85,B 0,C 180,E1 -14131.188,E2 -14131.188} C_VEL
LIN {X 0,Y 339.15,Z 470.785,A -85,B 0,C 180,E1 -14132.376,E2 -14132.376} C_VEL
LIN {X 0,Y 339.142,Z 469.511,A -85,B 0,C 180,E1 -14133.565,E2 -14133.565} C_VEL
LIN {X 0,Y 339.182,Z 467.737,A -85,B 0,C 180,E1 -14134.755,E2 -14134.755} C_VEL
LIN {X 0,Y 339.274,Z 464.044,A -85,B 0,C 180,E1 -14136.483,E2 -14136.483} C_VEL
LIN {X 0,Y 339.604,Z 458.662,A -85,B 0,C 180,E1 -14138.33,E2 -14138.33} C_VEL
LIN {X 0,Y 340.152,Z 451.779,A -85,B 0,C 180,E1 -14140.115,E2 -14140.115} C_VEL
LIN {X 0,Y 340.885,Z 444.272,A -85,B 0,C 180,E1 -14141.597,E2 -14141.597} C_VEL
LIN {X 0,Y 341.594,Z 436.873,A -85,B 0,C 180,E1 -14142.778,E2 -14142.778} C_VEL
LIN {X 0,Y 342.386,Z 428.958,A -85,B 0,C 180,E1 -14143.806,E2 -14143.806} C_VEL
LIN {X 0,Y 343.22,Z 420.601,A -85,B 0,C 180,E1 -14144.679,E2 -14144.679} C_VEL
LIN {X 0,Y 344.018,Z 409.918,A -85,B 0,C 180,E1 -14145.554,E2 -14145.554} C_VEL
LIN {X 0,Y 344.737,Z 398.283,A -85,B 0,C 180,E1 -14146.203,E2 -14146.203} C_VEL
LIN {X 0,Y 345.233,Z 388.524,A -85,B 0,C 180,E1 -14146.559,E2 -14146.559} C_VEL
LIN {X 0,Y 345.853,Z 345.435,A -85,B 0,C 180,E1 -14147.479,E2 -14147.479} C_VEL
LIN {X 0,Y 342.613,Z 319.328,A -85,B 0,C 180,E1 -14148.208,E2 -14148.208} C_VEL
LIN {X 0,Y 341.36,Z 310.364,A -85,B 0,C 180,E1 -14148.494,E2 -14148.494} C_VEL
LIN {X 0,Y 342.387,Z 297.905,A -85,B 0,C 180,E1 -14151.684,E2 -14151.684} C_VEL
LIN {X 0,Y 343.302,Z 287.047,A -85,B 0,C 180,E1 -14154.492,E2 -14154.492} C_VEL
LIN {X 0,Y 341.85,Z 278.436,A -85,B 0,C 180,E1 -14156.891,E2 -14156.891} C_VEL
LIN {X 0,Y 340.714,Z 272.855,A -85,B 0,C 180,E1 -14158.533,E2 -14158.533} C_VEL
LIN {X 0,Y 340.681,Z 272.858,A -85,B 0,C 180,E1 -14162.437,E2 -14162.437} C_VEL
LIN {X 0,Y 340.715,Z 272.858,A -85,B 0,C 180,E1 -14165.28,E2 -14165.28} C_VEL
LIN {X 0,Y 340.693,Z 272.857,A -85,B 0,C 180,E1 -14168.382,E2 -14168.382} C_VEL
LIN {X 0,Y 340.691,Z 272.857,A -85,B 0,C 180,E1 -14172.044,E2 -14172.044} C_VEL
LIN {X 0,Y 340.65,Z 272.863,A -85,B 0,C 180,E1 -14176.228,E2 -14176.228} C_VEL
LIN {X 0,Y 340.669,Z 272.865,A -85,B 0,C 180,E1 -14178.688,E2 -14178.688} C_VEL
LIN {X 0,Y 340.719,Z 272.853,A -85,B 0,C 180,E1 -14181.771,E2 -14181.771} C_VEL
LIN {X 0,Y 340.723,Z 272.853,A -85,B 0,C 180,E1 -14185.596,E2 -14185.596} C_VEL
LIN {X 0,Y 340.693,Z 272.857,A -85,B 0,C 180,E1 -14188.955,E2 -14188.955} C_VEL
LIN {X 0,Y 340.71,Z 272.855,A -85,B 0,C 180,E1 -14193.012,E2 -14193.012} C_VEL
LIN {X 0,Y 340.7,Z 272.856,A -85,B 0,C 180,E1 -14196.925,E2 -14196.925} C_VEL
LIN {X 0,Y 340.697,Z 272.856,A -85,B 0,C 180,E1 -14200.728,E2 -14200.728} C_VEL
LIN {X 0,Y 340.726,Z 272.852,A -85,B 0,C 180,E1 -14203.216,E2 -14203.216} C_VEL
LIN {X 0,Y 340.816,Z 272.841,A -85,B 0,C 180,E1 -14206.889,E2 -14206.889} C_VEL
LIN {X 0,Y 340.881,Z 272.832,A -85,B 0,C 180,E1 -14210.507,E2 -14210.507} C_VEL
LIN {X 0,Y 341.003,Z 272.816,A -85,B 0,C 180,E1 -14212.897,E2 -14212.897} C_VEL
LIN {X 0,Y 340.808,Z 272.844,A -85,B 0,C 180,E1 -14215.269,E2 -14215.269} C_VEL
LIN {X 0,Y 341.119,Z 272.808,A -85,B 0,C 180,E1 -14217.639,E2 -14217.639} C_VEL
LIN {X 0,Y 341.089,Z 272.81,A -85,B 0,C 180,E1 -14221.181,E2 -14221.181} C_VEL
LIN {X 0,Y 341.125,Z 272.801,A -85,B 0,C 180,E1 -14222.362,E2 -14222.362} C_VEL
LIN {X 0,Y 341.001,Z 272.822,A -85,B 0,C 180,E1 -14227.103,E2 -14227.103} C_VEL
LIN {X 0,Y 340.845,Z 272.839,A -85,B 0,C 180,E1 -14230.695,E2 -14230.695} C_VEL
LIN {X 0,Y 340.82,Z 272.84,A -85,B 0,C 180,E1 -14234.327,E2 -14234.327} C_VEL
LIN {X 0,Y 340.756,Z 272.85,A -85,B 0,C 180,E1 -14238.424,E2 -14238.424} C_VEL
LIN {X 0,Y 340.72,Z 272.853,A -85,B 0,C 180,E1 -14241.842,E2 -14241.842} C_VEL
LIN {X 0,Y 340.672,Z 272.859,A -85,B 0,C 180,E1 -14245.673,E2 -14245.673} C_VEL
LIN {X 0,Y 340.68,Z 272.861,A -85,B 0,C 180,E1 -14248.325,E2 -14248.325} C_VEL
LIN {X 0,Y 340.692,Z 272.857,A -85,B 0,C 180,E1 -14251.045,E2 -14251.045} C_VEL
LIN {X 0,Y 340.717,Z 272.852,A -85,B 0,C 180,E1 -14255.279,E2 -14255.279} C_VEL
LIN {X 0,Y 340.695,Z 272.861,A -85,B 0,C 180,E1 -14258.382,E2 -14258.382} C_VEL
LIN {X 0,Y 340.692,Z 272.861,A -85,B 0,C 180,E1 -14262.043,E2 -14262.043} C_VEL
LIN {X 0,Y 340.651,Z 272.866,A -85,B 0,C 180,E1 -14266.227,E2 -14266.227} C_VEL
LIN {X 0,Y 340.669,Z 272.859,A -85,B 0,C 180,E1 -14268.687,E2 -14268.687} C_VEL
LIN {X 0,Y 340.72,Z 272.855,A -85,B 0,C 180,E1 -14271.77,E2 -14271.77} C_VEL
LIN {X 0,Y 340.724,Z 272.856,A -85,B 0,C 180,E1 -14275.596,E2 -14275.596} C_VEL
LIN {X 0,Y 340.684,Z 272.858,A -85,B 0,C 180,E1 -14278.953,E2 -14278.953} C_VEL
LIN {X 0,Y 340.691,Z 272.857,A -85,B 0,C 180,E1 -14282.503,E2 -14282.503} C_VEL
LIN {X 0,Y 340.746,Z 272.854,A -85,B 0,C 180,E1 -14285.637,E2 -14285.637} C_VEL
LIN {X 0,Y 340.717,Z 272.86,A -85,B 0,C 180,E1 -14289.472,E2 -14289.472} C_VEL
LIN {X 0,Y 340.787,Z 272.959,A -85,B 0,C 180,E1 -14290.894,E2 -14290.894} C_VEL
LIN {X 0,Y 341.261,Z 275.333,A -85,B 0,C 180,E1 -14291.585,E2 -14291.585} C_VEL
LIN {X 0,Y 345.027,Z 287.471,A -85,B 0,C 180,E1 -14292.06,E2 -14292.06} C_VEL
LIN {X 0,Y 346.539,Z 295.282,A -85,B 0,C 180,E1 -14292.309,E2 -14292.309} C_VEL
LIN {X 0,Y 345.67,Z 351.711,A -85,B 0,C 180,E1 -14293.5,E2 -14293.5} C_VEL
LIN {X 0,Y 345.463,Z 360.699,A -85,B 0,C 180,E1 -14293.831,E2 -14293.831} C_VEL
LIN {X 0,Y 345.141,Z 370.224,A -85,B 0,C 180,E1 -14294.347,E2 -14294.347} C_VEL
LIN {X 0,Y 344.546,Z 380.219,A -85,B 0,C 180,E1 -14295.076,E2 -14295.076} C_VEL
LIN {X 0,Y 343.792,Z 390.578,A -85,B 0,C 180,E1 -14296.101,E2 -14296.101} C_VEL
LIN {X 0,Y 343.086,Z 398.688,A -85,B 0,C 180,E1 -14297.128,E2 -14297.128} C_VEL
LIN {X 0,Y 342.417,Z 405.376,A -85,B 0,C 180,E1 -14298.156,E2 -14298.156} C_VEL
LIN {X 0,Y 341.737,Z 411.706,A -85,B 0,C 180,E1 -14299.333,E2 -14299.333} C_VEL
LIN {X 0,Y 341.031,Z 418.129,A -85,B 0,C 180,E1 -14300.809,E2 -14300.809} C_VEL
LIN {X 0,Y 340.645,Z 422.374,A -85,B 0,C 180,E1 -14302.018,E2 -14302.018} C_VEL
LIN {X 0,Y 340.168,Z 426.506,A -85,B 0,C 180,E1 -14303.475,E2 -14303.475} C_VEL
LIN {X 0,Y 339.857,Z 429.154,A -85,B 0,C 180,E1 -14304.66,E2 -14304.66} C_VEL
LIN {X 0,Y 339.621,Z 432.046,A -85,B 0,C 180,E1 -14306.44,E2 -14306.44} C_VEL
LIN {X 0,Y 339.479,Z 433.312,A -85,B 0,C 180,E1 -14307.626,E2 -14307.626} C_VEL
LIN {X 0,Y 339.357,Z 434.114,A -85,B 0,C 180,E1 -14308.813,E2 -14308.813} C_VEL
LIN {X 0,Y 339.333,Z 434.418,A -85,B 0,C 180,E1 -14309.999,E2 -14309.999} C_VEL
LIN {X 0,Y 339.356,Z 434.143,A -85,B 0,C 180,E1 -14311.186,E2 -14311.186} C_VEL
LIN {X 0,Y 339.462,Z 433.4,A -85,B 0,C 180,E1 -14312.372,E2 -14312.372} C_VEL
LIN {X 0,Y 339.616,Z 432.192,A -85,B 0,C 180,E1 -14313.559,E2 -14313.559} C_VEL
LIN {X 0,Y 339.841,Z 429.361,A -85,B 0,C 180,E1 -14315.339,E2 -14315.339} C_VEL
LIN {X 0,Y 340.158,Z 426.778,A -85,B 0,C 180,E1 -14316.524,E2 -14316.524} C_VEL
LIN {X 0,Y 340.627,Z 422.781,A -85,B 0,C 180,E1 -14317.961,E2 -14317.961} C_VEL
LIN {X 0,Y 341.018,Z 418.553,A -85,B 0,C 180,E1 -14319.19,E2 -14319.19} C_VEL
LIN {X 0,Y 341.544,Z 413.627,A -85,B 0,C 180,E1 -14320.372,E2 -14320.372} C_VEL
LIN {X 0,Y 342.227,Z 407.674,A -85,B 0,C 180,E1 -14321.55,E2 -14321.55} C_VEL
LIN {X 0,Y 343.012,Z 400.423,A -85,B 0,C 180,E1 -14322.723,E2 -14322.723} C_VEL
LIN {X 0,Y 343.577,Z 393.899,A -85,B 0,C 180,E1 -14323.605,E2 -14323.605} C_VEL
LIN {X 0,Y 344.183,Z 385.994,A -85,B 0,C 180,E1 -14324.485,E2 -14324.485} C_VEL
LIN {X 0,Y 344.743,Z 377.822,A -85,B 0,C 180,E1 -14325.216,E2 -14325.216} C_VEL
LIN {X 0,Y 345.271,Z 369.533,A -85,B 0,C 180,E1 -14325.797,E2 -14325.797} C_VEL
LIN {X 0,Y 345.497,Z 360.582,A -85,B 0,C 180,E1 -14326.279,E2 -14326.279} C_VEL
LIN {X 0,Y 345.724,Z 351.122,A -85,B 0,C 180,E1 -14326.622,E2 -14326.622} C_VEL
LIN {X 0,Y 346.566,Z 295.289,A -85,B 0,C 180,E1 -14327.797,E2 -14327.797} C_VEL
LIN {X 0,Y 344.129,Z 283.921,A -85,B 0,C 180,E1 -14328.175,E2 -14328.175} C_VEL
LIN {X 0,Y 341.17,Z 275.083,A -85,B 0,C 180,E1 -14328.563,E2 -14328.563} C_VEL
LIN {X 0,Y 340.756,Z 272.857,A -85,B 0,C 180,E1 -14329.268,E2 -14329.268} C_VEL
LIN {X 0,Y 340.7,Z 272.857,A -85,B 0,C 180,E1 -14333.131,E2 -14333.131} C_VEL
LIN {X 0,Y 340.709,Z 272.856,A -85,B 0,C 180,E1 -14336.987,E2 -14336.987} C_VEL
LIN {X 0,Y 340.675,Z 272.862,A -85,B 0,C 180,E1 -14338.268,E2 -14338.268} C_VEL
LIN {X 0,Y 340.031,Z 272.949,A -85,B 0,C 180,E1 -14339.255,E2 -14339.255} C_VEL
LIN {X 0,Y 337.185,Z 273.305,A -85,B 0,C 180,E1 -14340.86,E2 -14340.86} C_VEL
LIN {X 0,Y 334.757,Z 273.601,A -85,B 0,C 180,E1 -14342.16,E2 -14342.16} C_VEL
LIN {X 0,Y 333.71,Z 273.726,A -85,B 0,C 180,E1 -14343.166,E2 -14343.166} C_VEL
LIN {X 0,Y 333.623,Z 273.735,A -85,B 0,C 180,E1 -14343.507,E2 -14343.507} C_VEL
LIN {X 0,Y 333.659,Z 273.733,A -85,B 0,C 180,E1 -14346.831,E2 -14346.831} C_VEL
LIN {X 0,Y 333.599,Z 273.739,A -85,B 0,C 180,E1 -14350.773,E2 -14350.773} C_VEL
LIN {X 0,Y 333.586,Z 273.745,A -85,B 0,C 180,E1 -14354.249,E2 -14354.249} C_VEL
LIN {X 0,Y 333.632,Z 273.738,A -85,B 0,C 180,E1 -14357.617,E2 -14357.617} C_VEL
LIN {X 0,Y 333.612,Z 273.739,A -85,B 0,C 180,E1 -14361.209,E2 -14361.209} C_VEL
LIN {X 0,Y 333.669,Z 273.735,A -85,B 0,C 180,E1 -14363.86,E2 -14363.86} C_VEL
LIN {X 0,Y 333.638,Z 273.739,A -85,B 0,C 180,E1 -14367.413,E2 -14367.413} C_VEL
LIN {X 0,Y 333.645,Z 273.736,A -85,B 0,C 180,E1 -14371.022,E2 -14371.022} C_VEL
LIN {X 0,Y 333.691,Z 273.732,A -85,B 0,C 180,E1 -14375.088,E2 -14375.088} C_VEL
LIN {X 0,Y 333.648,Z 273.737,A -85,B 0,C 180,E1 -14379.017,E2 -14379.017} C_VEL
LIN {X 0,Y 333.707,Z 273.728,A -85,B 0,C 180,E1 -14381.584,E2 -14381.584} C_VEL
LIN {X 0,Y 333.769,Z 273.718,A -85,B 0,C 180,E1 -14385.6,E2 -14385.6} C_VEL
LIN {X 0,Y 333.808,Z 273.718,A -85,B 0,C 180,E1 -14389.077,E2 -14389.077} C_VEL
LIN {X 0,Y 333.95,Z 273.701,A -85,B 0,C 180,E1 -14392.746,E2 -14392.746} C_VEL
LIN {X 0,Y 333.769,Z 273.718,A -85,B 0,C 180,E1 -14395.168,E2 -14395.168} C_VEL
LIN {X 0,Y 334.059,Z 273.681,A -85,B 0,C 180,E1 -14397.588,E2 -14397.588} C_VEL
LIN {X 0,Y 334.053,Z 273.684,A -85,B 0,C 180,E1 -14401.205,E2 -14401.205} C_VEL
LIN {X 0,Y 334.059,Z 273.687,A -85,B 0,C 180,E1 -14402.411,E2 -14402.411} C_VEL
LIN {X 0,Y 333.98,Z 273.694,A -85,B 0,C 180,E1 -14406.039,E2 -14406.039} C_VEL
LIN {X 0,Y 333.908,Z 273.706,A -85,B 0,C 180,E1 -14408.472,E2 -14408.472} C_VEL
LIN {X 0,Y 333.781,Z 273.722,A -85,B 0,C 180,E1 -14412.155,E2 -14412.155} C_VEL
LIN {X 0,Y 333.746,Z 273.723,A -85,B 0,C 180,E1 -14414.637,E2 -14414.637} C_VEL
LIN {X 0,Y 333.688,Z 273.73,A -85,B 0,C 180,E1 -14418.602,E2 -14418.602} C_VEL
LIN {X 0,Y 333.644,Z 273.737,A -85,B 0,C 180,E1 -14422.281,E2 -14422.281} C_VEL
LIN {X 0,Y 333.65,Z 273.734,A -85,B 0,C 180,E1 -14425.077,E2 -14425.077} C_VEL
LIN {X 0,Y 333.623,Z 273.738,A -85,B 0,C 180,E1 -14428.98,E2 -14428.98} C_VEL
LIN {X 0,Y 333.638,Z 273.735,A -85,B 0,C 180,E1 -14432.587,E2 -14432.587} C_VEL
LIN {X 0,Y 333.669,Z 273.732,A -85,B 0,C 180,E1 -14436.14,E2 -14436.14} C_VEL
LIN {X 0,Y 333.615,Z 273.742,A -85,B 0,C 180,E1 -14439.197,E2 -14439.197} C_VEL
LIN {X 0,Y 333.621,Z 273.738,A -85,B 0,C 180,E1 -14442.499,E2 -14442.499} C_VEL
LIN {X 0,Y 333.589,Z 273.742,A -85,B 0,C 180,E1 -14445.955,E2 -14445.955} C_VEL
LIN {X 0,Y 333.597,Z 273.744,A -85,B 0,C 180,E1 -14449.325,E2 -14449.325} C_VEL
LIN {X 0,Y 333.657,Z 273.737,A -85,B 0,C 180,E1 -14453.169,E2 -14453.169} C_VEL
LIN {X 0,Y 333.669,Z 273.733,A -85,B 0,C 180,E1 -14455.342,E2 -14455.342} C_VEL
LIN {X 0,Y 333.617,Z 273.739,A -85,B 0,C 180,E1 -14458.221,E2 -14458.221} C_VEL
LIN {X 0,Y 333.711,Z 273.892,A -85,B 0,C 180,E1 -14461.24,E2 -14461.24} C_VEL
LIN {X 0,Y 336.005,Z 285.692,A -85,B 0,C 180,E1 -14464.669,E2 -14464.669} C_VEL
LIN {X 0,Y 336.298,Z 289.139,A -85,B 0,C 180,E1 -14465.624,E2 -14465.624} C_VEL
LIN {X 0,Y 335,Z 303.591,A -85,B 0,C 180,E1 -14469.428,E2 -14469.428} C_VEL
LIN {X 0,Y 334.429,Z 310.039,A -85,B 0,C 180,E1 -14471.111,E2 -14471.111} C_VEL
LIN {X 0,Y 337.883,Z 335.064,A -85,B 0,C 180,E1 -14471.86,E2 -14471.86} C_VEL
LIN {X 0,Y 339.119,Z 347.848,A -85,B 0,C 180,E1 -14472.205,E2 -14472.205} C_VEL
LIN {X 0,Y 338.463,Z 388.768,A -85,B 0,C 180,E1 -14473.101,E2 -14473.101} C_VEL
LIN {X 0,Y 337.871,Z 399.959,A -85,B 0,C 180,E1 -14473.537,E2 -14473.537} C_VEL
LIN {X 0,Y 337.045,Z 411.677,A -85,B 0,C 180,E1 -14474.273,E2 -14474.273} C_VEL
LIN {X 0,Y 336.301,Z 420.386,A -85,B 0,C 180,E1 -14475.013,E2 -14475.013} C_VEL
LIN {X 0,Y 335.483,Z 428.71,A -85,B 0,C 180,E1 -14475.906,E2 -14475.906} C_VEL
LIN {X 0,Y 334.65,Z 436.595,A -85,B 0,C 180,E1 -14476.953,E2 -14476.953} C_VEL
LIN {X 0,Y 333.915,Z 443.977,A -85,B 0,C 180,E1 -14478.159,E2 -14478.159} C_VEL
LIN {X 0,Y 333.158,Z 451.473,A -85,B 0,C 180,E1 -14479.671,E2 -14479.671} C_VEL
LIN {X 0,Y 332.573,Z 458.328,A -85,B 0,C 180,E1 -14481.494,E2 -14481.494} C_VEL
LIN {X 0,Y 332.22,Z 463.542,A -85,B 0,C 180,E1 -14483.319,E2 -14483.319} C_VEL
LIN {X 0,Y 332.076,Z 467.377,A -85,B 0,C 180,E1 -14485.144,E2 -14485.144} C_VEL
LIN {X 0,Y 332.067,Z 469.143,A -85,B 0,C 180,E1 -14486.36,E2 -14486.36} C_VEL
LIN {X 0,Y 332.057,Z 470.407,A -85,B 0,C 180,E1 -14487.575,E2 -14487.575} C_VEL
LIN {X 0,Y 332.161,Z 471.199,A -85,B 0,C 180,E1 -14488.788,E2 -14488.788} C_VEL
LIN {X 0,Y 332.246,Z 471.5,A -85,B 0,C 180,E1 -14490.001,E2 -14490.001} C_VEL
LIN {X 0,Y 332.161,Z 471.194,A -85,B 0,C 180,E1 -14491.213,E2 -14491.213} C_VEL
LIN {X 0,Y 332.057,Z 470.393,A -85,B 0,C 180,E1 -14492.427,E2 -14492.427} C_VEL
LIN {X 0,Y 332.067,Z 469.119,A -85,B 0,C 180,E1 -14493.641,E2 -14493.641} C_VEL
LIN {X 0,Y 332.045,Z 466.204,A -85,B 0,C 180,E1 -14495.45,E2 -14495.45} C_VEL
LIN {X 0,Y 332.212,Z 463.497,A -85,B 0,C 180,E1 -14496.682,E2 -14496.682} C_VEL
LIN {X 0,Y 332.568,Z 458.268,A -85,B 0,C 180,E1 -14498.507,E2 -14498.507} C_VEL
LIN {X 0,Y 333.154,Z 451.384,A -85,B 0,C 180,E1 -14500.33,E2 -14500.33} C_VEL
LIN {X 0,Y 333.907,Z 443.876,A -85,B 0,C 180,E1 -14501.843,E2 -14501.843} C_VEL
LIN {X 0,Y 334.642,Z 436.476,A -85,B 0,C 180,E1 -14503.049,E2 -14503.049} C_VEL
LIN {X 0,Y 335.492,Z 428.562,A -85,B 0,C 180,E1 -14504.095,E2 -14504.095} C_VEL
LIN {X 0,Y 336.343,Z 420.204,A -85,B 0,C 180,E1 -14504.986,E2 -14504.986} C_VEL
LIN {X 0,Y 337.161,Z 409.519,A -85,B 0,C 180,E1 -14505.878,E2 -14505.878} C_VEL
LIN {X 0,Y 337.931,Z 397.882,A -85,B 0,C 180,E1 -14506.539,E2 -14506.539} C_VEL
LIN {X 0,Y 338.44,Z 388.117,A -85,B 0,C 180,E1 -14506.902,E2 -14506.902} C_VEL
LIN {X 0,Y 338.985,Z 345.129,A -85,B 0,C 180,E1 -14507.843,E2 -14507.843} C_VEL
LIN {X 0,Y 335.639,Z 318.42,A -85,B 0,C 180,E1 -14508.611,E2 -14508.611} C_VEL
LIN {X 0,Y 334.404,Z 310.014,A -85,B 0,C 180,E1 -14508.878,E2 -14508.878} C_VEL
LIN {X 0,Y 335.41,Z 298.705,A -85,B 0,C 180,E1 -14511.835,E2 -14511.835} C_VEL
LIN {X 0,Y 336.344,Z 289.064,A -85,B 0,C 180,E1 -14514.374,E2 -14514.374} C_VEL
LIN {X 0,Y 335.259,Z 281.697,A -85,B 0,C 180,E1 -14516.453,E2 -14516.453} C_VEL
LIN {X 0,Y 333.677,Z 273.733,A -85,B 0,C 180,E1 -14518.834,E2 -14518.834} C_VEL
LIN {X 0,Y 333.64,Z 273.735,A -85,B 0,C 180,E1 -14522.586,E2 -14522.586} C_VEL
LIN {X 0,Y 333.673,Z 273.731,A -85,B 0,C 180,E1 -14526.14,E2 -14526.14} C_VEL
LIN {X 0,Y 333.62,Z 273.741,A -85,B 0,C 180,E1 -14529.197,E2 -14529.197} C_VEL
LIN {X 0,Y 333.627,Z 273.739,A -85,B 0,C 180,E1 -14532.499,E2 -14532.499} C_VEL
LIN {X 0,Y 333.594,Z 273.741,A -85,B 0,C 180,E1 -14535.955,E2 -14535.955} C_VEL
LIN {X 0,Y 333.602,Z 273.741,A -85,B 0,C 180,E1 -14539.325,E2 -14539.325} C_VEL
LIN {X 0,Y 333.662,Z 273.733,A -85,B 0,C 180,E1 -14543.169,E2 -14543.169} C_VEL
LIN {X 0,Y 333.673,Z 273.731,A -85,B 0,C 180,E1 -14545.341,E2 -14545.341} C_VEL
LIN {X 0,Y 333.63,Z 273.74,A -85,B 0,C 180,E1 -14548.222,E2 -14548.222} C_VEL
LIN {X 0,Y 333.629,Z 273.737,A -85,B 0,C 180,E1 -14551.02,E2 -14551.02} C_VEL
LIN {X 0,Y 333.656,Z 273.733,A -85,B 0,C 180,E1 -14554.923,E2 -14554.923} C_VEL
LIN {X 0,Y 333.649,Z 273.734,A -85,B 0,C 180,E1 -14559.017,E2 -14559.017} C_VEL
LIN {X 0,Y 333.706,Z 273.729,A -85,B 0,C 180,E1 -14561.585,E2 -14561.585} C_VEL
LIN {X 0,Y 333.76,Z 273.723,A -85,B 0,C 180,E1 -14565.611,E2 -14565.611} C_VEL
LIN {X 0,Y 333.81,Z 273.714,A -85,B 0,C 180,E1 -14569.077,E2 -14569.077} C_VEL
LIN {X 0,Y 333.958,Z 273.692,A -85,B 0,C 180,E1 -14572.746,E2 -14572.746} C_VEL
LIN {X 0,Y 333.775,Z 273.719,A -85,B 0,C 180,E1 -14575.169,E2 -14575.169} C_VEL
LIN {X 0,Y 334.059,Z 273.688,A -85,B 0,C 180,E1 -14577.589,E2 -14577.589} C_VEL
LIN {X 0,Y 334.06,Z 273.686,A -85,B 0,C 180,E1 -14581.206,E2 -14581.206} C_VEL
LIN {X 0,Y 334.065,Z 273.68,A -85,B 0,C 180,E1 -14582.412,E2 -14582.412} C_VEL
LIN {X 0,Y 333.959,Z 273.694,A -85,B 0,C 180,E1 -14586.469,E2 -14586.469} C_VEL
LIN {X 0,Y 333.82,Z 273.714,A -85,B 0,C 180,E1 -14589.696,E2 -14589.696} C_VEL
LIN {X 0,Y 333.787,Z 273.717,A -85,B 0,C 180,E1 -14593.392,E2 -14593.392} C_VEL
LIN {X 0,Y 333.681,Z 273.733,A -85,B 0,C 180,E1 -14597.15,E2 -14597.15} C_VEL
LIN {X 0,Y 333.637,Z 273.735,A -85,B 0,C 180,E1 -14599.697,E2 -14599.697} C_VEL
LIN {X 0,Y 333.651,Z 273.735,A -85,B 0,C 180,E1 -14602.281,E2 -14602.281} C_VEL
LIN {X 0,Y 333.66,Z 273.735,A -85,B 0,C 180,E1 -14605.078,E2 -14605.078} C_VEL
LIN {X 0,Y 333.652,Z 273.735,A -85,B 0,C 180,E1 -14608.978,E2 -14608.978} C_VEL
LIN {X 0,Y 333.645,Z 273.738,A -85,B 0,C 180,E1 -14612.586,E2 -14612.586} C_VEL
LIN {X 0,Y 333.675,Z 273.732,A -85,B 0,C 180,E1 -14616.139,E2 -14616.139} C_VEL
LIN {X 0,Y 333.603,Z 273.74,A -85,B 0,C 180,E1 -14619.199,E2 -14619.199} C_VEL
LIN {X 0,Y 333.628,Z 273.738,A -85,B 0,C 180,E1 -14622.498,E2 -14622.498} C_VEL
LIN {X 0,Y 333.595,Z 273.745,A -85,B 0,C 180,E1 -14625.954,E2 -14625.954} C_VEL
LIN {X 0,Y 333.603,Z 273.739,A -85,B 0,C 180,E1 -14629.324,E2 -14629.324} C_VEL
LIN {X 0,Y 333.664,Z 273.73,A -85,B 0,C 180,E1 -14633.168,E2 -14633.168} C_VEL
LIN {X 0,Y 333.675,Z 273.732,A -85,B 0,C 180,E1 -14635.341,E2 -14635.341} C_VEL
LIN {X 0,Y 333.622,Z 273.738,A -85,B 0,C 180,E1 -14638.221,E2 -14638.221} C_VEL
LIN {X 0,Y 333.631,Z 273.737,A -85,B 0,C 180,E1 -14641.02,E2 -14641.02} C_VEL
LIN {X 0,Y 333.698,Z 273.731,A -85,B 0,C 180,E1 -14645.088,E2 -14645.088} C_VEL
LIN {X 0,Y 333.656,Z 273.737,A -85,B 0,C 180,E1 -14649.017,E2 -14649.017} C_VEL
LIN {X 0,Y 333.754,Z 273.924,A -85,B 0,C 180,E1 -14650.645,E2 -14650.645} C_VEL
LIN {X 0,Y 334.13,Z 275.75,A -85,B 0,C 180,E1 -14651.177,E2 -14651.177} C_VEL
LIN {X 0,Y 338.356,Z 288.695,A -85,B 0,C 180,E1 -14651.711,E2 -14651.711} C_VEL
LIN {X 0,Y 339.812,Z 297.357,A -85,B 0,C 180,E1 -14651.983,E2 -14651.983} C_VEL
LIN {X 0,Y 338.892,Z 352.119,A -85,B 0,C 180,E1 -14653.16,E2 -14653.16} C_VEL
LIN {X 0,Y 338.677,Z 361.1,A -85,B 0,C 180,E1 -14653.498,E2 -14653.498} C_VEL
LIN {X 0,Y 338.344,Z 370.623,A -85,B 0,C 180,E1 -14654.024,E2 -14654.024} C_VEL
LIN {X 0,Y 337.724,Z 380.615,A -85,B 0,C 180,E1 -14654.768,E2 -14654.768} C_VEL
LIN {X 0,Y 337,Z 389.725,A -85,B 0,C 180,E1 -14655.661,E2 -14655.661} C_VEL
LIN {X 0,Y 336.192,Z 399.082,A -85,B 0,C 180,E1 -14656.859,E2 -14656.859} C_VEL
LIN {X 0,Y 335.495,Z 405.77,A -85,B 0,C 180,E1 -14657.907,E2 -14657.907} C_VEL
LIN {X 0,Y 334.783,Z 412.1,A -85,B 0,C 180,E1 -14659.109,E2 -14659.109} C_VEL
LIN {X 0,Y 334.054,Z 418.522,A -85,B 0,C 180,E1 -14660.616,E2 -14660.616} C_VEL
LIN {X 0,Y 333.602,Z 423.088,A -85,B 0,C 180,E1 -14661.952,E2 -14661.952} C_VEL
LIN {X 0,Y 333.142,Z 426.898,A -85,B 0,C 180,E1 -14663.336,E2 -14663.336} C_VEL
LIN {X 0,Y 332.805,Z 429.546,A -85,B 0,C 180,E1 -14664.546,E2 -14664.546} C_VEL
LIN {X 0,Y 332.542,Z 432.438,A -85,B 0,C 180,E1 -14666.364,E2 -14666.364} C_VEL
LIN {X 0,Y 332.395,Z 433.704,A -85,B 0,C 180,E1 -14667.576,E2 -14667.576} C_VEL
LIN {X 0,Y 332.282,Z 434.505,A -85,B 0,C 180,E1 -14668.787,E2 -14668.787} C_VEL
LIN {X 0,Y 332.254,Z 434.809,A -85,B 0,C 180,E1 -14669.999,E2 -14669.999} C_VEL
LIN {X 0,Y 332.281,Z 434.534,A -85,B 0,C 180,E1 -14671.211,E2 -14671.211} C_VEL
LIN {X 0,Y 332.378,Z 433.791,A -85,B 0,C 180,E1 -14672.423,E2 -14672.423} C_VEL
LIN {X 0,Y 332.536,Z 432.583,A -85,B 0,C 180,E1 -14673.635,E2 -14673.635} C_VEL
LIN {X 0,Y 332.788,Z 429.752,A -85,B 0,C 180,E1 -14675.453,E2 -14675.453} C_VEL
LIN {X 0,Y 333.139,Z 427.167,A -85,B 0,C 180,E1 -14676.662,E2 -14676.662} C_VEL
LIN {X 0,Y 333.559,Z 423.593,A -85,B 0,C 180,E1 -14677.995,E2 -14677.995} C_VEL
LIN {X 0,Y 334.033,Z 418.942,A -85,B 0,C 180,E1 -14679.384,E2 -14679.384} C_VEL
LIN {X 0,Y 334.566,Z 414.016,A -85,B 0,C 180,E1 -14680.591,E2 -14680.591} C_VEL
LIN {X 0,Y 335.303,Z 408.061,A -85,B 0,C 180,E1 -14681.791,E2 -14681.791} C_VEL
LIN {X 0,Y 336.107,Z 400.811,A -85,B 0,C 180,E1 -14682.989,E2 -14682.989} C_VEL
LIN {X 0,Y 336.706,Z 394.286,A -85,B 0,C 180,E1 -14683.888,E2 -14683.888} C_VEL
LIN {X 0,Y 337.338,Z 386.379,A -85,B 0,C 180,E1 -14684.785,E2 -14684.785} C_VEL
LIN {X 0,Y 337.931,Z 378.206,A -85,B 0,C 180,E1 -14685.53,E2 -14685.53} C_VEL
LIN {X 0,Y 338.465,Z 369.915,A -85,B 0,C 180,E1 -14686.124,E2 -14686.124} C_VEL
LIN {X 0,Y 338.716,Z 360.961,A -85,B 0,C 180,E1 -14686.615,E2 -14686.615} C_VEL
LIN {X 0,Y 338.94,Z 351.645,A -85,B 0,C 180,E1 -14686.96,E2 -14686.96} C_VEL
LIN {X 0,Y 339.762,Z 295.924,A -85,B 0,C 180,E1 -14688.16,E2 -14688.16} C_VEL
LIN {X 0,Y 337.608,Z 285.973,A -85,B 0,C 180,E1 -14688.501,E2 -14688.501} C_VEL
LIN {X 0,Y 334.061,Z 275.525,A -85,B 0,C 180,E1 -14688.96,E2 -14688.96} C_VEL
LIN {X 0,Y 333.711,Z 273.735,A -85,B 0,C 180,E1 -14689.559,E2 -14689.559} C_VEL
LIN {X 0,Y 333.643,Z 273.735,A -85,B 0,C 180,E1 -14693.591,E2 -14693.591} C_VEL
LIN {X 0,Y 333.658,Z 273.733,A -85,B 0,C 180,E1 -14697.606,E2 -14697.606} C_VEL
LIN {X 0,Y 333.652,Z 273.739,A -85,B 0,C 180,E1 -14700.366,E2 -14700.366} C_VEL
LIN {X 0,Y 333.623,Z 273.735,A -85,B 0,C 180,E1 -14703.507,E2 -14703.507} C_VEL
LIN {X 0,Y 332.949,Z 273.824,A -85,B 0,C 180,E1 -14704.516,E2 -14704.516} C_VEL
LIN {X 0,Y 330.089,Z 274.181,A -85,B 0,C 180,E1 -14706.156,E2 -14706.156} C_VEL
LIN {X 0,Y 327.673,Z 274.483,A -85,B 0,C 180,E1 -14707.485,E2 -14707.485} C_VEL
LIN {X 0,Y 326.642,Z 274.61,A -85,B 0,C 180,E1 -14708.514,E2 -14708.514} C_VEL
LIN {X 0,Y 326.562,Z 274.617,A -85,B 0,C 180,E1 -14708.863,E2 -14708.863} C_VEL
LIN {X 0,Y 326.568,Z 274.615,A -85,B 0,C 180,E1 -14712.97,E2 -14712.97} C_VEL
LIN {X 0,Y 326.568,Z 274.614,A -85,B 0,C 180,E1 -14717.028,E2 -14717.028} C_VEL
LIN {X 0,Y 326.567,Z 274.615,A -85,B 0,C 180,E1 -14720.781,E2 -14720.781} C_VEL
LIN {X 0,Y 326.606,Z 274.611,A -85,B 0,C 180,E1 -14724.479,E2 -14724.479} C_VEL
LIN {X 0,Y 326.603,Z 274.615,A -85,B 0,C 180,E1 -14727.455,E2 -14727.455} C_VEL
LIN {X 0,Y 326.584,Z 274.614,A -85,B 0,C 180,E1 -14730.333,E2 -14730.333} C_VEL
LIN {X 0,Y 326.629,Z 274.608,A -85,B 0,C 180,E1 -14734.511,E2 -14734.511} C_VEL
LIN {X 0,Y 326.604,Z 274.611,A -85,B 0,C 180,E1 -14738.542,E2 -14738.542} C_VEL
LIN {X 0,Y 326.643,Z 274.611,A -85,B 0,C 180,E1 -14741.206,E2 -14741.206} C_VEL
LIN {X 0,Y 326.72,Z 274.596,A -85,B 0,C 180,E1 -14745.459,E2 -14745.459} C_VEL
LIN {X 0,Y 326.749,Z 274.597,A -85,B 0,C 180,E1 -14748.838,E2 -14748.838} C_VEL
LIN {X 0,Y 326.907,Z 274.577,A -85,B 0,C 180,E1 -14752.589,E2 -14752.589} C_VEL
LIN {X 0,Y 326.739,Z 274.593,A -85,B 0,C 180,E1 -14755.064,E2 -14755.064} C_VEL
LIN {X 0,Y 327.002,Z 274.559,A -85,B 0,C 180,E1 -14757.536,E2 -14757.536} C_VEL
LIN {X 0,Y 327.023,Z 274.56,A -85,B 0,C 180,E1 -14761.231,E2 -14761.231} C_VEL
LIN {X 0,Y 326.742,Z 274.594,A -85,B 0,C 180,E1 -14763.7,E2 -14763.7} C_VEL
LIN {X 0,Y 326.934,Z 274.573,A -85,B 0,C 180,E1 -14766.17,E2 -14766.17} C_VEL
LIN {X 0,Y 326.776,Z 274.592,A -85,B 0,C 180,E1 -14769.907,E2 -14769.907} C_VEL
LIN {X 0,Y 326.737,Z 274.596,A -85,B 0,C 180,E1 -14773.686,E2 -14773.686} C_VEL
LIN {X 0,Y 326.622,Z 274.61,A -85,B 0,C 180,E1 -14777.532,E2 -14777.532} C_VEL
LIN {X 0,Y 326.601,Z 274.613,A -85,B 0,C 180,E1 -14781.458,E2 -14781.458} C_VEL
LIN {X 0,Y 326.593,Z 274.615,A -85,B 0,C 180,E1 -14785.492,E2 -14785.492} C_VEL
LIN {X 0,Y 326.584,Z 274.615,A -85,B 0,C 180,E1 -14788.257,E2 -14788.257} C_VEL
LIN {X 0,Y 326.567,Z 274.618,A -85,B 0,C 180,E1 -14791.098,E2 -14791.098} C_VEL
LIN {X 0,Y 326.602,Z 274.614,A -85,B 0,C 180,E1 -14794.02,E2 -14794.02} C_VEL
LIN {X 0,Y 326.617,Z 274.614,A -85,B 0,C 180,E1 -14797.238,E2 -14797.238} C_VEL
LIN {X 0,Y 326.539,Z 274.624,A -85,B 0,C 180,E1 -14801.125,E2 -14801.125} C_VEL
LIN {X 0,Y 326.554,Z 274.621,A -85,B 0,C 180,E1 -14803.527,E2 -14803.527} C_VEL
LIN {X 0,Y 326.567,Z 274.621,A -85,B 0,C 180,E1 -14807.03,E2 -14807.03} C_VEL
LIN {X 0,Y 326.577,Z 274.617,A -85,B 0,C 180,E1 -14811.386,E2 -14811.386} C_VEL
LIN {X 0,Y 326.614,Z 274.615,A -85,B 0,C 180,E1 -14814.852,E2 -14814.852} C_VEL
LIN {X 0,Y 326.601,Z 274.613,A -85,B 0,C 180,E1 -14817.456,E2 -14817.456} C_VEL
LIN {X 0,Y 326.667,Z 274.707,A -85,B 0,C 180,E1 -14820.918,E2 -14820.918} C_VEL
LIN {X 0,Y 328.9,Z 286.138,A -85,B 0,C 180,E1 -14824.324,E2 -14824.324} C_VEL
LIN {X 0,Y 329.33,Z 289.945,A -85,B 0,C 180,E1 -14825.41,E2 -14825.41} C_VEL
LIN {X 0,Y 328.322,Z 300.788,A -85,B 0,C 180,E1 -14828.331,E2 -14828.331} C_VEL
LIN {X 0,Y 327.534,Z 309.587,A -85,B 0,C 180,E1 -14830.683,E2 -14830.683} C_VEL
LIN {X 0,Y 331.168,Z 336.077,A -85,B 0,C 180,E1 -14831.51,E2 -14831.51} C_VEL
LIN {X 0,Y 332.364,Z 348.291,A -85,B 0,C 180,E1 -14831.849,E2 -14831.849} C_VEL
LIN {X 0,Y 331.655,Z 388.39,A -85,B 0,C 180,E1 -14832.743,E2 -14832.743} C_VEL
LIN {X 0,Y 331.061,Z 399.576,A -85,B 0,C 180,E1 -14833.188,E2 -14833.188} C_VEL
LIN {X 0,Y 330.194,Z 411.289,A -85,B 0,C 180,E1 -14833.938,E2 -14833.938} C_VEL
LIN {X 0,Y 329.434,Z 419.998,A -85,B 0,C 180,E1 -14834.693,E2 -14834.693} C_VEL
LIN {X 0,Y 328.608,Z 428.322,A -85,B 0,C 180,E1 -14835.604,E2 -14835.604} C_VEL
LIN {X 0,Y 327.738,Z 436.206,A -85,B 0,C 180,E1 -14836.673,E2 -14836.673} C_VEL
LIN {X 0,Y 326.927,Z 443.586,A -85,B 0,C 180,E1 -14837.902,E2 -14837.902} C_VEL
LIN {X 0,Y 326.141,Z 451.081,A -85,B 0,C 180,E1 -14839.446,E2 -14839.446} C_VEL
LIN {X 0,Y 325.513,Z 457.935,A -85,B 0,C 180,E1 -14841.308,E2 -14841.308} C_VEL
LIN {X 0,Y 325.141,Z 463.15,A -85,B 0,C 180,E1 -14843.173,E2 -14843.173} C_VEL
LIN {X 0,Y 324.974,Z 466.985,A -85,B 0,C 180,E1 -14845.038,E2 -14845.038} C_VEL
LIN {X 0,Y 324.991,Z 468.753,A -85,B 0,C 180,E1 -14846.281,E2 -14846.281} C_VEL
LIN {X 0,Y 324.968,Z 470.016,A -85,B 0,C 180,E1 -14847.522,E2 -14847.522} C_VEL
LIN {X 0,Y 325.064,Z 470.807,A -85,B 0,C 180,E1 -14848.762,E2 -14848.762} C_VEL
LIN {X 0,Y 325.169,Z 471.109,A -85,B 0,C 180,E1 -14850.001,E2 -14850.001} C_VEL
LIN {X 0,Y 325.064,Z 470.802,A -85,B 0,C 180,E1 -14851.239,E2 -14851.239} C_VEL
LIN {X 0,Y 324.969,Z 470.001,A -85,B 0,C 180,E1 -14852.48,E2 -14852.48} C_VEL
LIN {X 0,Y 324.992,Z 468.727,A -85,B 0,C 180,E1 -14853.72,E2 -14853.72} C_VEL
LIN {X 0,Y 324.974,Z 466.948,A -85,B 0,C 180,E1 -14854.963,E2 -14854.963} C_VEL
LIN {X 0,Y 325.137,Z 463.102,A -85,B 0,C 180,E1 -14856.828,E2 -14856.828} C_VEL
LIN {X 0,Y 325.51,Z 457.872,A -85,B 0,C 180,E1 -14858.693,E2 -14858.693} C_VEL
LIN {X 0,Y 326.137,Z 450.988,A -85,B 0,C 180,E1 -14860.555,E2 -14860.555} C_VEL
LIN {X 0,Y 326.918,Z 443.479,A -85,B 0,C 180,E1 -14862.1,E2 -14862.1} C_VEL
LIN {X 0,Y 327.729,Z 436.081,A -85,B 0,C 180,E1 -14863.329,E2 -14863.329} C_VEL
LIN {X 0,Y 328.616,Z 428.167,A -85,B 0,C 180,E1 -14864.396,E2 -14864.396} C_VEL
LIN {X 0,Y 329.485,Z 419.808,A -85,B 0,C 180,E1 -14865.306,E2 -14865.306} C_VEL
LIN {X 0,Y 330.343,Z 409.121,A -85,B 0,C 180,E1 -14866.215,E2 -14866.215} C_VEL
LIN {X 0,Y 331.131,Z 397.48,A -85,B 0,C 180,E1 -14866.889,E2 -14866.889} C_VEL
LIN {X 0,Y 331.659,Z 387.71,A -85,B 0,C 180,E1 -14867.258,E2 -14867.258} C_VEL
LIN {X 0,Y 332.239,Z 346.028,A -85,B 0,C 180,E1 -14868.189,E2 -14868.189} C_VEL
LIN {X 0,Y 328.913,Z 319.282,A -85,B 0,C 180,E1 -14868.977,E2 -14868.977} C_VEL
LIN {X 0,Y 327.466,Z 309.594,A -85,B 0,C 180,E1 -14869.298,E2 -14869.298} C_VEL
LIN {X 0,Y 328.551,Z 298.302,A -85,B 0,C 180,E1 -14872.315,E2 -14872.315} C_VEL
LIN {X 0,Y 329.368,Z 289.863,A -85,B 0,C 180,E1 -14874.588,E2 -14874.588} C_VEL
LIN {X 0,Y 328.217,Z 282.494,A -85,B 0,C 180,E1 -14876.723,E2 -14876.723} C_VEL
LIN {X 0,Y 326.662,Z 274.607,A -85,B 0,C 180,E1 -14879.128,E2 -14879.128} C_VEL
LIN {X 0,Y 326.615,Z 274.613,A -85,B 0,C 180,E1 -14882.945,E2 -14882.945} C_VEL
LIN {X 0,Y 326.61,Z 274.613,A -85,B 0,C 180,E1 -14885.52,E2 -14885.52} C_VEL
LIN {X 0,Y 326.588,Z 274.617,A -85,B 0,C 180,E1 -14889.222,E2 -14889.222} C_VEL
LIN {X 0,Y 326.572,Z 274.621,A -85,B 0,C 180,E1 -14892.971,E2 -14892.971} C_VEL
LIN {X 0,Y 326.572,Z 274.619,A -85,B 0,C 180,E1 -14897.03,E2 -14897.03} C_VEL
LIN {X 0,Y 326.587,Z 274.618,A -85,B 0,C 180,E1 -14900.779,E2 -14900.779} C_VEL
LIN {X 0,Y 326.611,Z 274.616,A -85,B 0,C 180,E1 -14904.48,E2 -14904.48} C_VEL
LIN {X 0,Y 326.609,Z 274.611,A -85,B 0,C 180,E1 -14907.456,E2 -14907.456} C_VEL
LIN {X 0,Y 326.58,Z 274.62,A -85,B 0,C 180,E1 -14910.333,E2 -14910.333} C_VEL
LIN {X 0,Y 326.595,Z 274.613,A -85,B 0,C 180,E1 -14913.135,E2 -14913.135} C_VEL
LIN {X 0,Y 326.592,Z 274.613,A -85,B 0,C 180,E1 -14917.211,E2 -14917.211} C_VEL
LIN {X 0,Y 326.629,Z 274.608,A -85,B 0,C 180,E1 -14921.217,E2 -14921.217} C_VEL
LIN {X 0,Y 326.716,Z 274.599,A -85,B 0,C 180,E1 -14925.467,E2 -14925.467} C_VEL
LIN {X 0,Y 326.75,Z 274.592,A -85,B 0,C 180,E1 -14928.838,E2 -14928.838} C_VEL
LIN {X 0,Y 326.915,Z 274.569,A -85,B 0,C 180,E1 -14932.589,E2 -14932.589} C_VEL
LIN {X 0,Y 326.745,Z 274.594,A -85,B 0,C 180,E1 -14935.065,E2 -14935.065} C_VEL
LIN {X 0,Y 327.002,Z 274.567,A -85,B 0,C 180,E1 -14937.537,E2 -14937.537} C_VEL
LIN {X 0,Y 327.03,Z 274.561,A -85,B 0,C 180,E1 -14941.232,E2 -14941.232} C_VEL
LIN {X 0,Y 326.747,Z 274.592,A -85,B 0,C 180,E1 -14943.7,E2 -14943.7} C_VEL
LIN {X 0,Y 326.921,Z 274.57,A -85,B 0,C 180,E1 -14946.457,E2 -14946.457} C_VEL
LIN {X 0,Y 326.783,Z 274.589,A -85,B 0,C 180,E1 -14949.907,E2 -14949.907} C_VEL
LIN {X 0,Y 326.744,Z 274.592,A -85,B 0,C 180,E1 -14953.686,E2 -14953.686} C_VEL
LIN {X 0,Y 326.629,Z 274.608,A -85,B 0,C 180,E1 -14957.532,E2 -14957.532} C_VEL
LIN {X 0,Y 326.604,Z 274.612,A -85,B 0,C 180,E1 -14961.458,E2 -14961.458} C_VEL
LIN {X 0,Y 326.602,Z 274.612,A -85,B 0,C 180,E1 -14965.491,E2 -14965.491} C_VEL
LIN {X 0,Y 326.597,Z 274.614,A -85,B 0,C 180,E1 -14968.256,E2 -14968.256} C_VEL
LIN {X 0,Y 326.573,Z 274.616,A -85,B 0,C 180,E1 -14971.097,E2 -14971.097} C_VEL
LIN {X 0,Y 326.608,Z 274.611,A -85,B 0,C 180,E1 -14974.019,E2 -14974.019} C_VEL
LIN {X 0,Y 326.624,Z 274.609,A -85,B 0,C 180,E1 -14977.237,E2 -14977.237} C_VEL
LIN {X 0,Y 326.544,Z 274.618,A -85,B 0,C 180,E1 -14981.124,E2 -14981.124} C_VEL
LIN {X 0,Y 326.56,Z 274.616,A -85,B 0,C 180,E1 -14983.526,E2 -14983.526} C_VEL
LIN {X 0,Y 326.573,Z 274.616,A -85,B 0,C 180,E1 -14987.029,E2 -14987.029} C_VEL
LIN {X 0,Y 326.573,Z 274.61,A -85,B 0,C 180,E1 -14990.781,E2 -14990.781} C_VEL
LIN {X 0,Y 326.612,Z 274.61,A -85,B 0,C 180,E1 -14994.48,E2 -14994.48} C_VEL
LIN {X 0,Y 326.606,Z 274.614,A -85,B 0,C 180,E1 -14997.455,E2 -14997.455} C_VEL
LIN {X 0,Y 326.58,Z 274.615,A -85,B 0,C 180,E1 -15000.332,E2 -15000.332} C_VEL
LIN {X 0,Y 326.608,Z 274.613,A -85,B 0,C 180,E1 -15003.135,E2 -15003.135} C_VEL
LIN {X 0,Y 326.633,Z 274.612,A -85,B 0,C 180,E1 -15005.869,E2 -15005.869} C_VEL
LIN {X 0,Y 326.627,Z 274.616,A -85,B 0,C 180,E1 -15009.862,E2 -15009.862} C_VEL
LIN {X 0,Y 326.698,Z 274.798,A -85,B 0,C 180,E1 -15010.357,E2 -15010.357} C_VEL
LIN {X 0,Y 326.94,Z 275.936,A -85,B 0,C 180,E1 -15010.726,E2 -15010.726} C_VEL
LIN {X 0,Y 331.81,Z 290.586,A -85,B 0,C 180,E1 -15011.371,E2 -15011.371} C_VEL
LIN {X 0,Y 333.096,Z 297.842,A -85,B 0,C 180,E1 -15011.609,E2 -15011.609} C_VEL
LIN {X 0,Y 332.126,Z 352.528,A -85,B 0,C 180,E1 -15012.807,E2 -15012.807} C_VEL
LIN {X 0,Y 331.902,Z 361.502,A -85,B 0,C 180,E1 -15013.152,E2 -15013.152} C_VEL
LIN {X 0,Y 331.556,Z 371.021,A -85,B 0,C 180,E1 -15013.688,E2 -15013.688} C_VEL
LIN {X 0,Y 330.903,Z 381.012,A -85,B 0,C 180,E1 -15014.446,E2 -15014.446} C_VEL
LIN {X 0,Y 330.144,Z 390.121,A -85,B 0,C 180,E1 -15015.357,E2 -15015.357} C_VEL
LIN {X 0,Y 329.297,Z 399.477,A -85,B 0,C 180,E1 -15016.579,E2 -15016.579} C_VEL
LIN {X 0,Y 328.587,Z 406.163,A -85,B 0,C 180,E1 -15017.649,E2 -15017.649} C_VEL
LIN {X 0,Y 327.843,Z 412.493,A -85,B 0,C 180,E1 -15018.875,E2 -15018.875} C_VEL
LIN {X 0,Y 327.054,Z 418.915,A -85,B 0,C 180,E1 -15020.413,E2 -15020.413} C_VEL
LIN {X 0,Y 326.55,Z 423.84,A -85,B 0,C 180,E1 -15021.895,E2 -15021.895} C_VEL
LIN {X 0,Y 325.922,Z 428.769,A -85,B 0,C 180,E1 -15023.81,E2 -15023.81} C_VEL
LIN {X 0,Y 325.626,Z 431.078,A -85,B 0,C 180,E1 -15025.047,E2 -15025.047} C_VEL
LIN {X 0,Y 325.463,Z 432.831,A -85,B 0,C 180,E1 -15026.285,E2 -15026.285} C_VEL
LIN {X 0,Y 325.312,Z 434.096,A -85,B 0,C 180,E1 -15027.523,E2 -15027.523} C_VEL
LIN {X 0,Y 325.209,Z 434.896,A -85,B 0,C 180,E1 -15028.761,E2 -15028.761} C_VEL
LIN {X 0,Y 325.179,Z 435.2,A -85,B 0,C 180,E1 -15029.999,E2 -15029.999} C_VEL
LIN {X 0,Y 325.208,Z 434.924,A -85,B 0,C 180,E1 -15031.238,E2 -15031.238} C_VEL
LIN {X 0,Y 325.295,Z 434.182,A -85,B 0,C 180,E1 -15032.476,E2 -15032.476} C_VEL
LIN {X 0,Y 325.457,Z 432.974,A -85,B 0,C 180,E1 -15033.714,E2 -15033.714} C_VEL
LIN {X 0,Y 325.741,Z 430.141,A -85,B 0,C 180,E1 -15035.571,E2 -15035.571} C_VEL
LIN {X 0,Y 326.119,Z 427.556,A -85,B 0,C 180,E1 -15036.806,E2 -15036.806} C_VEL
LIN {X 0,Y 326.74,Z 422.473,A -85,B 0,C 180,E1 -15038.659,E2 -15038.659} C_VEL
LIN {X 0,Y 327.305,Z 417.006,A -85,B 0,C 180,E1 -15040.203,E2 -15040.203} C_VEL
LIN {X 0,Y 328.168,Z 410.123,A -85,B 0,C 180,E1 -15041.738,E2 -15041.738} C_VEL
LIN {X 0,Y 329.087,Z 402.214,A -85,B 0,C 180,E1 -15043.114,E2 -15043.114} C_VEL
LIN {X 0,Y 329.833,Z 394.673,A -85,B 0,C 180,E1 -15044.183,E2 -15044.183} C_VEL
LIN {X 0,Y 330.339,Z 388.261,A -85,B 0,C 180,E1 -15044.948,E2 -15044.948} C_VEL
LIN {X 0,Y 331.015,Z 380.455,A -85,B 0,C 180,E1 -15045.705,E2 -15045.705} C_VEL
LIN {X 0,Y 331.584,Z 371.505,A -85,B 0,C 180,E1 -15046.389,E2 -15046.389} C_VEL
LIN {X 0,Y 331.939,Z 362.168,A -85,B 0,C 180,E1 -15046.924,E2 -15046.924} C_VEL
LIN {X 0,Y 332.148,Z 353.071,A -85,B 0,C 180,E1 -15047.285,E2 -15047.285} C_VEL
LIN {X 0,Y 333.108,Z 297.308,A -85,B 0,C 180,E1 -15048.513,E2 -15048.513} C_VEL
LIN {X 0,Y 331.05,Z 287.927,A -85,B 0,C 180,E1 -15048.845,E2 -15048.845} C_VEL
LIN {X 0,Y 326.91,Z 275.91,A -85,B 0,C 180,E1 -15049.398,E2 -15049.398} C_VEL
LIN {X 0,Y 326.618,Z 274.616,A -85,B 0,C 180,E1 -15049.897,E2 -15049.897} C_VEL
LIN {X 0,Y 326.591,Z 274.619,A -85,B 0,C 180,E1 -15052.789,E2 -15052.789} C_VEL
LIN {X 0,Y 326.595,Z 274.616,A -85,B 0,C 180,E1 -15056.865,E2 -15056.865} C_VEL
LIN {X 0,Y 326.606,Z 274.615,A -85,B 0,C 180,E1 -15060.601,E2 -15060.601} C_VEL
LIN {X 0,Y 326.603,Z 274.614,A -85,B 0,C 180,E1 -15064.019,E2 -15064.019} C_VEL
LIN {X 0,Y 326.62,Z 274.609,A -85,B 0,C 180,E1 -15067.236,E2 -15067.236} C_VEL
LIN {X 0,Y 326.562,Z 274.617,A -85,B 0,C 180,E1 -15068.863,E2 -15068.863} C_VEL
LIN {X 0,Y 325.898,Z 274.703,A -85,B 0,C 180,E1 -15069.891,E2 -15069.891} C_VEL
LIN {X 0,Y 323.031,Z 275.056,A -85,B 0,C 180,E1 -15071.565,E2 -15071.565} C_VEL
LIN {X 0,Y 320.599,Z 275.359,A -85,B 0,C 180,E1 -15072.921,E2 -15072.921} C_VEL
LIN {X 0,Y 319.558,Z 275.494,A -85,B 0,C 180,E1 -15073.971,E2 -15073.971} C_VEL
LIN {X 0,Y 319.475,Z 275.497,A -85,B 0,C 180,E1 -15074.327,E2 -15074.327} C_VEL
LIN {X 0,Y 319.546,Z 275.489,A -85,B 0,C 180,E1 -15077.015,E2 -15077.015} C_VEL
LIN {X 0,Y 319.511,Z 275.496,A -85,B 0,C 180,E1 -15080.365,E2 -15080.365} C_VEL
LIN {X 0,Y 319.574,Z 275.487,A -85,B 0,C 180,E1 -15084.457,E2 -15084.457} C_VEL
LIN {X 0,Y 319.518,Z 275.494,A -85,B 0,C 180,E1 -15088.137,E2 -15088.137} C_VEL
LIN {X 0,Y 319.563,Z 275.491,A -85,B 0,C 180,E1 -15091.604,E2 -15091.604} C_VEL
LIN {X 0,Y 319.568,Z 275.493,A -85,B 0,C 180,E1 -15095.301,E2 -15095.301} C_VEL
LIN {X 0,Y 319.559,Z 275.489,A -85,B 0,C 180,E1 -15098.045,E2 -15098.045} C_VEL
LIN {X 0,Y 319.581,Z 275.485,A -85,B 0,C 180,E1 -15102.068,E2 -15102.068} C_VEL
LIN {X 0,Y 319.704,Z 275.467,A -85,B 0,C 180,E1 -15106.006,E2 -15106.006} C_VEL
LIN {X 0,Y 319.728,Z 275.468,A -85,B 0,C 180,E1 -15109.872,E2 -15109.872} C_VEL
LIN {X 0,Y 319.892,Z 275.446,A -85,B 0,C 180,E1 -15113.693,E2 -15113.693} C_VEL
LIN {X 0,Y 319.948,Z 275.437,A -85,B 0,C 180,E1 -15117.482,E2 -15117.482} C_VEL
LIN {X 0,Y 319.992,Z 275.435,A -85,B 0,C 180,E1 -15121.258,E2 -15121.258} C_VEL
LIN {X 0,Y 319.692,Z 275.472,A -85,B 0,C 180,E1 -15123.781,E2 -15123.781} C_VEL
LIN {X 0,Y 319.892,Z 275.451,A -85,B 0,C 180,E1 -15126.307,E2 -15126.307} C_VEL
LIN {X 0,Y 319.728,Z 275.472,A -85,B 0,C 180,E1 -15130.128,E2 -15130.128} C_VEL
LIN {X 0,Y 319.704,Z 275.475,A -85,B 0,C 180,E1 -15133.993,E2 -15133.993} C_VEL
LIN {X 0,Y 319.578,Z 275.491,A -85,B 0,C 180,E1 -15137.931,E2 -15137.931} C_VEL
LIN {X 0,Y 319.556,Z 275.495,A -85,B 0,C 180,E1 -15141.955,E2 -15141.955} C_VEL
LIN {X 0,Y 319.543,Z 275.494,A -85,B 0,C 180,E1 -15146.096,E2 -15146.096} C_VEL
LIN {X 0,Y 319.519,Z 275.495,A -85,B 0,C 180,E1 -15148.94,E2 -15148.94} C_VEL
LIN {X 0,Y 319.519,Z 275.498,A -85,B 0,C 180,E1 -15151.863,E2 -15151.863} C_VEL
LIN {X 0,Y 319.575,Z 275.493,A -85,B 0,C 180,E1 -15155.543,E2 -15155.543} C_VEL
LIN {X 0,Y 319.523,Z 275.497,A -85,B 0,C 180,E1 -15159.662,E2 -15159.662} C_VEL
LIN {X 0,Y 319.514,Z 275.499,A -85,B 0,C 180,E1 -15163.46,E2 -15163.46} C_VEL
LIN {X 0,Y 319.546,Z 275.496,A -85,B 0,C 180,E1 -15167.016,E2 -15167.016} C_VEL
LIN {X 0,Y 319.541,Z 275.492,A -85,B 0,C 180,E1 -15170.371,E2 -15170.371} C_VEL
LIN {X 0,Y 319.574,Z 275.489,A -85,B 0,C 180,E1 -15174.458,E2 -15174.458} C_VEL
LIN {X 0,Y 319.516,Z 275.495,A -85,B 0,C 180,E1 -15178.137,E2 -15178.137} C_VEL
LIN {X 0,Y 319.627,Z 275.654,A -85,B 0,C 180,E1 -15180.62,E2 -15180.62} C_VEL
LIN {X 0,Y 321.864,Z 287.071,A -85,B 0,C 180,E1 -15184.107,E2 -15184.107} C_VEL
LIN {X 0,Y 322.348,Z 291.959,A -85,B 0,C 180,E1 -15185.529,E2 -15185.529} C_VEL
LIN {X 0,Y 320.797,Z 307.511,A -85,B 0,C 180,E1 -15189.794,E2 -15189.794} C_VEL
LIN {X 0,Y 320.617,Z 309.25,A -85,B 0,C 180,E1 -15190.268,E2 -15190.268} C_VEL
LIN {X 0,Y 324.47,Z 337.143,A -85,B 0,C 180,E1 -15191.147,E2 -15191.147} C_VEL
LIN {X 0,Y 325.613,Z 348.704,A -85,B 0,C 180,E1 -15191.477,E2 -15191.477} C_VEL
LIN {X 0,Y 324.927,Z 386.847,A -85,B 0,C 180,E1 -15192.338,E2 -15192.338} C_VEL
LIN {X 0,Y 324.486,Z 395.868,A -85,B 0,C 180,E1 -15192.675,E2 -15192.675} C_VEL
LIN {X 0,Y 323.832,Z 405.505,A -85,B 0,C 180,E1 -15193.208,E2 -15193.208} C_VEL
LIN {X 0,Y 323.044,Z 414.657,A -85,B 0,C 180,E1 -15193.897,E2 -15193.897} C_VEL
LIN {X 0,Y 322.036,Z 425.466,A -85,B 0,C 180,E1 -15194.981,E2 -15194.981} C_VEL
LIN {X 0,Y 321.075,Z 433.766,A -85,B 0,C 180,E1 -15196.068,E2 -15196.068} C_VEL
LIN {X 0,Y 320.155,Z 441.48,A -85,B 0,C 180,E1 -15197.32,E2 -15197.32} C_VEL
LIN {X 0,Y 319.463,Z 447.84,A -85,B 0,C 180,E1 -15198.581,E2 -15198.581} C_VEL
LIN {X 0,Y 318.874,Z 453.127,A -85,B 0,C 180,E1 -15199.845,E2 -15199.845} C_VEL
LIN {X 0,Y 318.459,Z 457.543,A -85,B 0,C 180,E1 -15201.114,E2 -15201.114} C_VEL
LIN {X 0,Y 318.077,Z 462.758,A -85,B 0,C 180,E1 -15203.021,E2 -15203.021} C_VEL
LIN {X 0,Y 317.883,Z 466.592,A -85,B 0,C 180,E1 -15204.927,E2 -15204.927} C_VEL
LIN {X 0,Y 317.916,Z 468.362,A -85,B 0,C 180,E1 -15206.198,E2 -15206.198} C_VEL
LIN {X 0,Y 317.883,Z 469.625,A -85,B 0,C 180,E1 -15207.466,E2 -15207.466} C_VEL
LIN {X 0,Y 317.968,Z 470.415,A -85,B 0,C 180,E1 -15208.734,E2 -15208.734} C_VEL
LIN {X 0,Y 318.078,Z 470.717,A -85,B 0,C 180,E1 -15210.001,E2 -15210.001} C_VEL
LIN {X 0,Y 317.968,Z 470.41,A -85,B 0,C 180,E1 -15211.267,E2 -15211.267} C_VEL
LIN {X 0,Y 317.883,Z 469.609,A -85,B 0,C 180,E1 -15212.535,E2 -15212.535} C_VEL
LIN {X 0,Y 317.917,Z 468.335,A -85,B 0,C 180,E1 -15213.803,E2 -15213.803} C_VEL
LIN {X 0,Y 317.886,Z 466.554,A -85,B 0,C 180,E1 -15215.074,E2 -15215.074} C_VEL
LIN {X 0,Y 318.074,Z 462.708,A -85,B 0,C 180,E1 -15216.981,E2 -15216.981} C_VEL
LIN {X 0,Y 318.457,Z 457.477,A -85,B 0,C 180,E1 -15218.887,E2 -15218.887} C_VEL
LIN {X 0,Y 319.121,Z 450.592,A -85,B 0,C 180,E1 -15220.79,E2 -15220.79} C_VEL
LIN {X 0,Y 319.955,Z 443.083,A -85,B 0,C 180,E1 -15222.367,E2 -15222.367} C_VEL
LIN {X 0,Y 320.82,Z 435.686,A -85,B 0,C 180,E1 -15223.621,E2 -15223.621} C_VEL
LIN {X 0,Y 321.754,Z 427.772,A -85,B 0,C 180,E1 -15224.71,E2 -15224.71} C_VEL
LIN {X 0,Y 322.626,Z 419.41,A -85,B 0,C 180,E1 -15225.639,E2 -15225.639} C_VEL
LIN {X 0,Y 323.544,Z 408.724,A -85,B 0,C 180,E1 -15226.565,E2 -15226.565} C_VEL
LIN {X 0,Y 324.347,Z 397.079,A -85,B 0,C 180,E1 -15227.253,E2 -15227.253} C_VEL
LIN {X 0,Y 324.892,Z 387.304,A -85,B 0,C 180,E1 -15227.629,E2 -15227.629} C_VEL
LIN {X 0,Y 325.498,Z 346.749,A -85,B 0,C 180,E1 -15228.553,E2 -15228.553} C_VEL
LIN {X 0,Y 322.328,Z 321.101,A -85,B 0,C 180,E1 -15229.329,E2 -15229.329} C_VEL
LIN {X 0,Y 320.597,Z 309.172,A -85,B 0,C 180,E1 -15229.735,E2 -15229.735} C_VEL
LIN {X 0,Y 321.68,Z 297.895,A -85,B 0,C 180,E1 -15232.818,E2 -15232.818} C_VEL
LIN {X 0,Y 322.377,Z 290.66,A -85,B 0,C 180,E1 -15234.814,E2 -15234.814} C_VEL
LIN {X 0,Y 320.663,Z 280.914,A -85,B 0,C 180,E1 -15237.731,E2 -15237.731} C_VEL
LIN {X 0,Y 319.596,Z 275.486,A -85,B 0,C 180,E1 -15239.475,E2 -15239.475} C_VEL
LIN {X 0,Y 319.577,Z 275.49,A -85,B 0,C 180,E1 -15243.353,E2 -15243.353} C_VEL
LIN {X 0,Y 319.555,Z 275.491,A -85,B 0,C 180,E1 -15246.429,E2 -15246.429} C_VEL
LIN {X 0,Y 319.529,Z 275.494,A -85,B 0,C 180,E1 -15249.662,E2 -15249.662} C_VEL
LIN {X 0,Y 319.519,Z 275.496,A -85,B 0,C 180,E1 -15253.46,E2 -15253.46} C_VEL
LIN {X 0,Y 319.551,Z 275.494,A -85,B 0,C 180,E1 -15257.016,E2 -15257.016} C_VEL
LIN {X 0,Y 319.531,Z 275.496,A -85,B 0,C 180,E1 -15260.369,E2 -15260.369} C_VEL
LIN {X 0,Y 319.579,Z 275.492,A -85,B 0,C 180,E1 -15264.458,E2 -15264.458} C_VEL
LIN {X 0,Y 319.525,Z 275.496,A -85,B 0,C 180,E1 -15268.138,E2 -15268.138} C_VEL
LIN {X 0,Y 319.544,Z 275.491,A -85,B 0,C 180,E1 -15271.613,E2 -15271.613} C_VEL
LIN {X 0,Y 319.525,Z 275.493,A -85,B 0,C 180,E1 -15275.298,E2 -15275.298} C_VEL
LIN {X 0,Y 319.563,Z 275.494,A -85,B 0,C 180,E1 -15278.045,E2 -15278.045} C_VEL
LIN {X 0,Y 319.575,Z 275.492,A -85,B 0,C 180,E1 -15282.068,E2 -15282.068} C_VEL
LIN {X 0,Y 319.695,Z 275.476,A -85,B 0,C 180,E1 -15286.006,E2 -15286.006} C_VEL
LIN {X 0,Y 319.733,Z 275.468,A -85,B 0,C 180,E1 -15289.872,E2 -15289.872} C_VEL
LIN {X 0,Y 319.899,Z 275.448,A -85,B 0,C 180,E1 -15293.694,E2 -15293.694} C_VEL
LIN {X 0,Y 319.949,Z 275.445,A -85,B 0,C 180,E1 -15297.482,E2 -15297.482} C_VEL
LIN {X 0,Y 319.999,Z 275.437,A -85,B 0,C 180,E1 -15301.259,E2 -15301.259} C_VEL
LIN {X 0,Y 319.697,Z 275.469,A -85,B 0,C 180,E1 -15303.782,E2 -15303.782} C_VEL
LIN {X 0,Y 319.887,Z 275.446,A -85,B 0,C 180,E1 -15306.438,E2 -15306.438} C_VEL
LIN {X 0,Y 319.735,Z 275.467,A -85,B 0,C 180,E1 -15310.128,E2 -15310.128} C_VEL
LIN {X 0,Y 319.711,Z 275.466,A -85,B 0,C 180,E1 -15313.993,E2 -15313.993} C_VEL
LIN {X 0,Y 319.58,Z 275.485,A -85,B 0,C 180,E1 -15317.932,E2 -15317.932} C_VEL
LIN {X 0,Y 319.562,Z 275.488,A -85,B 0,C 180,E1 -15321.955,E2 -15321.955} C_VEL
LIN {X 0,Y 319.551,Z 275.491,A -85,B 0,C 180,E1 -15326.096,E2 -15326.096} C_VEL
LIN {X 0,Y 319.532,Z 275.494,A -85,B 0,C 180,E1 -15328.939,E2 -15328.939} C_VEL
LIN {X 0,Y 319.525,Z 275.494,A -85,B 0,C 180,E1 -15331.863,E2 -15331.863} C_VEL
LIN {X 0,Y 319.58,Z 275.483,A -85,B 0,C 180,E1 -15335.542,E2 -15335.542} C_VEL
LIN {X 0,Y 319.53,Z 275.494,A -85,B 0,C 180,E1 -15339.662,E2 -15339.662} C_VEL
LIN {X 0,Y 319.52,Z 275.493,A -85,B 0,C 180,E1 -15343.46,E2 -15343.46} C_VEL
LIN {X 0,Y 319.552,Z 275.491,A -85,B 0,C 180,E1 -15347.015,E2 -15347.015} C_VEL
LIN {X 0,Y 319.516,Z 275.49,A -85,B 0,C 180,E1 -15350.366,E2 -15350.366} C_VEL
LIN {X 0,Y 319.58,Z 275.486,A -85,B 0,C 180,E1 -15354.457,E2 -15354.457} C_VEL
LIN {X 0,Y 319.521,Z 275.496,A -85,B 0,C 180,E1 -15358.136,E2 -15358.136} C_VEL
LIN {X 0,Y 319.546,Z 275.496,A -85,B 0,C 180,E1 -15361.612,E2 -15361.612} C_VEL
